LIN {X 0.311,Y -645.263,Z 996.603,A 0.000,B 0.000,C 90.000,E1 324.482} C_DIS
LIN {X 0.129,Y -646.144,Z 996.595,A 0.000,B 0.000,C 90.000,E1 323.004} C_DIS
LIN {X -0.105,Y -646.582,Z 996.589,A 0.000,B 0.000,C 90.000,E1 322.029} C_DIS
LIN {X 0.123,Y -647.178,Z 996.581,A 0.000,B 0.000,C 90.000,E1 320.517} C_DIS
LIN {X -0.362,Y -648.118,Z 996.568,A 0.000,B 0.000,C 90.000,E1 318.324} C_DIS
LIN {X 0.227,Y -649.121,Z 996.560,A 0.000,B 0.000,C 90.000,E1 316.782} C_DIS
LIN {X -0.160,Y -650.130,Z 996.550,A 0.000,B 0.000,C 90.000,E1 315.081} C_DIS
LIN {X -0.098,Y -651.626,Z 996.539,A 0.000,B 0.000,C 90.000,E1 313.095} C_DIS
LIN {X 0.087,Y -652.642,Z 996.531,A 0.000,B 0.000,C 90.000,E1 311.595} C_DIS
LIN {X -0.104,Y -653.353,Z 996.524,A 0.000,B 0.000,C 90.000,E1 310.378} C_DIS
LIN {X -0.253,Y -654.049,Z 996.516,A 0.000,B 0.000,C 90.000,E1 308.910} C_DIS
LIN {X -0.386,Y -654.669,Z 996.508,A 0.000,B 0.000,C 90.000,E1 307.443} C_DIS
LIN {X 0.072,Y -654.916,Z 996.504,A 0.000,B 0.000,C 90.000,E1 306.664} C_DIS
LIN {X 0.085,Y -655.183,Z 996.496,A 0.000,B 0.000,C 90.000,E1 305.185} C_DIS
LIN {X 0.192,Y -655.481,Z 996.486,A 0.000,B 0.000,C 90.000,E1 303.452} C_DIS
LIN {X 0.053,Y -661.224,Z 996.451,A 0.000,B 0.000,C 90.000,E1 297.078} C_DIS
LIN {X -0.315,Y -664.130,Z 996.440,A 0.000,B 0.000,C 90.000,E1 295.155} C_DIS
LIN {X -0.012,Y -665.464,Z 996.434,A 0.000,B 0.000,C 90.000,E1 294.155} C_DIS
LIN {X -0.299,Y -666.631,Z 996.429,A 0.000,B 0.000,C 90.000,E1 293.206} C_DIS
LIN {X -0.114,Y -667.165,Z 996.425,A 0.000,B 0.000,C 90.000,E1 292.461} C_DIS
LIN {X -0.071,Y -667.271,Z 996.422,A 0.000,B 0.000,C 90.000,E1 291.972} C_DIS
LIN {X 0.220,Y -666.897,Z 996.419,A 0.000,B 0.000,C 90.000,E1 291.461} C_DIS
LIN {X 0.120,Y -666.527,Z 996.418,A 0.000,B 0.000,C 90.000,E1 291.227} C_DIS
LIN {X 0.260,Y -665.623,Z 996.417,A 0.000,B 0.000,C 90.000,E1 290.972} C_DIS
LIN {X 0.229,Y -664.050,Z 996.415,A 0.000,B 0.000,C 90.000,E1 290.610} C_DIS
LIN {X 0.296,Y -663.310,Z 996.414,A 0.000,B 0.000,C 90.000,E1 290.482} C_DIS
LIN {X 0.127,Y -662.192,Z 996.413,A 0.000,B 0.000,C 90.000,E1 290.375} C_DIS
LIN {X 0.079,Y -657.367,Z 996.411,A 0.000,B 0.000,C 90.000,E1 289.939} C_DIS
LIN {X 0.198,Y -655.675,Z 996.410,A 0.000,B 0.000,C 90.000,E1 289.812} C_DIS
LIN {X 0.177,Y -647.687,Z 996.408,A 0.000,B 0.000,C 90.000,E1 289.341} C_DIS
LIN {X -0.198,Y -644.564,Z 996.407,A 0.000,B 0.000,C 90.000,E1 289.195} C_DIS
LIN {X -0.301,Y -640.203,Z 996.405,A 0.000,B 0.000,C 90.000,E1 288.906} C_DIS
LIN {X -0.336,Y -640.181,Z 996.405,A 0.000,B 0.000,C 90.000,E1 288.906} C_DIS
LIN {X -0.088,Y -640.114,Z 996.405,A 0.000,B 0.000,C 90.000,E1 288.833} C_DIS
LIN {X 0.205,Y -641.641,Z 996.402,A 0.000,B 0.000,C 90.000,E1 288.417} C_DIS
LIN {X -0.250,Y -649.985,Z 996.395,A 0.000,B 0.000,C 90.000,E1 287.094} C_DIS
LIN {X 0.135,Y -653.488,Z 996.391,A 0.000,B 0.000,C 90.000,E1 286.441} C_DIS
LIN {X -0.107,Y -655.841,Z 996.389,A 0.000,B 0.000,C 90.000,E1 285.969} C_DIS
LIN {X -0.046,Y -656.935,Z 996.387,A 0.000,B 0.000,C 90.000,E1 285.717} C_DIS
LIN {X -0.271,Y -658.778,Z 996.385,A 0.000,B 0.000,C 90.000,E1 285.245} C_DIS
LIN {X 0.258,Y -659.581,Z 996.383,A 0.000,B 0.000,C 90.000,E1 284.954} C_DIS
LIN {X 0.054,Y -660.892,Z 996.381,A 0.000,B 0.000,C 90.000,E1 284.481} C_DIS
LIN {X -0.234,Y -662.248,Z 996.376,A 0.000,B 0.000,C 90.000,E1 283.772} C_DIS
LIN {X 0.226,Y -662.891,Z 996.374,A 0.000,B 0.000,C 90.000,E1 283.244} C_DIS
LIN {X -0.045,Y -663.382,Z 996.370,A 0.000,B 0.000,C 90.000,E1 282.535} C_DIS
LIN {X 0.333,Y -663.486,Z 996.366,A 0.000,B 0.000,C 90.000,E1 281.771} C_DIS
LIN {X 0.149,Y -663.317,Z 996.363,A 0.000,B 0.000,C 90.000,E1 281.299} C_DIS
LIN {X -0.258,Y -662.702,Z 996.359,A 0.000,B 0.000,C 90.000,E1 280.602} C_DIS
LIN {X 0.200,Y -661.947,Z 996.356,A 0.000,B 0.000,C 90.000,E1 280.074} C_DIS
LIN {X -0.114,Y -660.970,Z 996.353,A 0.000,B 0.000,C 90.000,E1 279.613} C_DIS
LIN {X -0.218,Y -660.446,Z 996.352,A 0.000,B 0.000,C 90.000,E1 279.378} C_DIS
LIN {X 0.113,Y -658.986,Z 996.349,A 0.000,B 0.000,C 90.000,E1 278.859} C_DIS
LIN {X -0.211,Y -657.223,Z 996.347,A 0.000,B 0.000,C 90.000,E1 278.398} C_DIS
LIN {X 0.197,Y -655.123,Z 996.344,A 0.000,B 0.000,C 90.000,E1 277.871} C_DIS
LIN {X -0.127,Y -653.259,Z 996.342,A 0.000,B 0.000,C 90.000,E1 277.530} C_DIS
LIN {X 0.274,Y -651.156,Z 996.340,A 0.000,B 0.000,C 90.000,E1 277.125} C_DIS
LIN {X -0.098,Y -647.850,Z 996.337,A 0.000,B 0.000,C 90.000,E1 276.663} C_DIS
LIN {X 0.051,Y -643.017,Z 996.334,A 0.000,B 0.000,C 90.000,E1 276.030} C_DIS
LIN {X 0.267,Y -638.641,Z 996.331,A 0.000,B 0.000,C 90.000,E1 275.511} C_DIS
LIN {X -0.240,Y -632.519,Z 996.327,A 0.000,B 0.000,C 90.000,E1 274.935} C_DIS
LIN {X 0.180,Y -627.269,Z 996.325,A 0.000,B 0.000,C 90.000,E1 274.416} C_DIS
LIN {X 0.190,Y -618.735,Z 996.321,A 0.000,B 0.000,C 90.000,E1 273.726} C_DIS
LIN {X 0.131,Y -611.173,Z 996.318,A 0.000,B 0.000,C 90.000,E1 273.212} C_DIS
LIN {X -0.225,Y -604.977,Z 996.316,A 0.000,B 0.000,C 90.000,E1 272.865} C_DIS
LIN {X 0.210,Y -598.422,Z 996.314,A 0.000,B 0.000,C 90.000,E1 272.465} C_DIS
LIN {X -0.129,Y -591.494,Z 996.312,A 0.000,B 0.000,C 90.000,E1 272.178} C_DIS
LIN {X 0.053,Y -584.129,Z 996.311,A 0.000,B 0.000,C 90.000,E1 271.892} C_DIS
LIN {X 0.222,Y -576.582,Z 996.309,A 0.000,B 0.000,C 90.000,E1 271.661} C_DIS
LIN {X -0.030,Y -570.873,Z 996.309,A 0.000,B 0.000,C 90.000,E1 271.547} C_DIS
LIN {X -0.069,Y -564.513,Z 996.308,A 0.000,B 0.000,C 90.000,E1 271.432} C_DIS
LIN {X 0.029,Y -558.252,Z 996.308,A 0.000,B 0.000,C 90.000,E1 271.375} C_DIS
LIN {X -0.014,Y -543.150,Z 996.308,A 0.000,B 0.000,C 90.000,E1 271.375} C_DIS
LIN {X 0.138,Y -542.514,Z 996.305,A 0.000,B 0.000,C 90.000,E1 270.917} C_DIS
LIN {X 0.065,Y -540.998,Z 996.293,A 0.000,B 0.000,C 90.000,E1 268.797} C_DIS
LIN {X 0.187,Y -540.032,Z 996.286,A 0.000,B 0.000,C 90.000,E1 267.364} C_DIS
LIN {X -0.262,Y -539.190,Z 996.279,A 0.000,B 0.000,C 90.000,E1 266.274} C_DIS
LIN {X -0.088,Y -537.915,Z 996.270,A 0.000,B 0.000,C 90.000,E1 264.546} C_DIS
LIN {X 0.007,Y -536.641,Z 996.262,A 0.000,B 0.000,C 90.000,E1 263.109} C_DIS
LIN {X 0.179,Y -534.965,Z 996.252,A 0.000,B 0.000,C 90.000,E1 261.376} C_DIS
LIN {X -0.133,Y -533.227,Z 996.243,A 0.000,B 0.000,C 90.000,E1 259.690} C_DIS
LIN {X 0.183,Y -531.087,Z 996.232,A 0.000,B 0.000,C 90.000,E1 257.645} C_DIS
LIN {X 0.036,Y -528.840,Z 996.220,A 0.000,B 0.000,C 90.000,E1 255.644} C_DIS
LIN {X 0.126,Y -525.952,Z 996.206,A 0.000,B 0.000,C 90.000,E1 253.032} C_DIS
LIN {X 0.117,Y -524.641,Z 996.199,A 0.000,B 0.000,C 90.000,E1 251.873} C_DIS
LIN {X -0.069,Y -523.224,Z 996.193,A 0.000,B 0.000,C 90.000,E1 250.732} C_DIS
LIN {X 0.205,Y -521.009,Z 996.183,A 0.000,B 0.000,C 90.000,E1 248.954} C_DIS
LIN {X -0.054,Y -518.737,Z 996.174,A 0.000,B 0.000,C 90.000,E1 247.230} C_DIS
LIN {X -0.105,Y -517.539,Z 996.169,A 0.000,B 0.000,C 90.000,E1 246.357} C_DIS
LIN {X 0.305,Y -515.339,Z 996.160,A 0.000,B 0.000,C 90.000,E1 244.845} C_DIS
LIN {X 0.092,Y -513.544,Z 996.154,A 0.000,B 0.000,C 90.000,E1 243.691} C_DIS
LIN {X -0.059,Y -510.285,Z 996.142,A 0.000,B 0.000,C 90.000,E1 241.641} C_DIS
LIN {X 0.221,Y -507.774,Z 996.134,A 0.000,B 0.000,C 90.000,E1 240.127} C_DIS
LIN {X 0.129,Y -505.635,Z 996.128,A 0.000,B 0.000,C 90.000,E1 238.948} C_DIS
LIN {X 0.142,Y -502.701,Z 996.119,A 0.000,B 0.000,C 90.000,E1 237.454} C_DIS
LIN {X -0.193,Y -500.193,Z 996.113,A 0.000,B 0.000,C 90.000,E1 236.294} C_DIS
LIN {X 0.126,Y -497.517,Z 996.106,A 0.000,B 0.000,C 90.000,E1 235.055} C_DIS
LIN {X -0.272,Y -495.439,Z 996.101,A 0.000,B 0.000,C 90.000,E1 234.196} C_DIS
LIN {X 0.108,Y -491.665,Z 996.093,A 0.000,B 0.000,C 90.000,E1 232.637} C_DIS
LIN {X -0.008,Y -486.585,Z 996.081,A 0.000,B 0.000,C 90.000,E1 230.517} C_DIS
LIN {X 0.001,Y -481.585,Z 996.069,A 0.000,B 0.000,C 90.000,E1 228.366} C_DIS
LIN {X 0.107,Y -475.618,Z 996.053,A 0.000,B 0.000,C 90.000,E1 225.567} C_DIS
LIN {X -0.146,Y -473.022,Z 996.046,A 0.000,B 0.000,C 90.000,E1 224.352} C_DIS
LIN {X -0.011,Y -469.581,Z 996.038,A 0.000,B 0.000,C 90.000,E1 222.771} C_DIS
LIN {X 0.155,Y -465.426,Z 996.027,A 0.000,B 0.000,C 90.000,E1 220.862} C_DIS
LIN {X 0.024,Y -463.299,Z 996.022,A 0.000,B 0.000,C 90.000,E1 219.930} C_DIS
LIN {X 0.066,Y -459.757,Z 996.013,A 0.000,B 0.000,C 90.000,E1 218.338} C_DIS
LIN {X 0.052,Y -455.563,Z 996.002,A 0.000,B 0.000,C 90.000,E1 216.423} C_DIS
LIN {X 0.130,Y -451.324,Z 995.992,A 0.000,B 0.000,C 90.000,E1 214.485} C_DIS
LIN {X 0.040,Y -447.850,Z 995.983,A 0.000,B 0.000,C 90.000,E1 212.880} C_DIS
LIN {X 0.072,Y -443.624,Z 995.972,A 0.000,B 0.000,C 90.000,E1 210.924} C_DIS
LIN {X 0.116,Y -440.040,Z 995.963,A 0.000,B 0.000,C 90.000,E1 209.283} C_DIS
LIN {X -0.048,Y -434.074,Z 995.948,A 0.000,B 0.000,C 90.000,E1 206.668} C_DIS
LIN {X -0.198,Y -430.307,Z 995.939,A 0.000,B 0.000,C 90.000,E1 205.027} C_DIS
LIN {X 0.131,Y -425.028,Z 995.926,A 0.000,B 0.000,C 90.000,E1 202.642} C_DIS
LIN {X 0.026,Y -421.297,Z 995.917,A 0.000,B 0.000,C 90.000,E1 200.972} C_DIS
LIN {X 0.092,Y -417.787,Z 995.907,A 0.000,B 0.000,C 90.000,E1 199.268} C_DIS
LIN {X -0.144,Y -413.191,Z 995.894,A 0.000,B 0.000,C 90.000,E1 196.913} C_DIS
LIN {X -0.092,Y -410.150,Z 995.884,A 0.000,B 0.000,C 90.000,E1 195.190} C_DIS
LIN {X -0.092,Y -406.672,Z 995.873,A 0.000,B 0.000,C 90.000,E1 193.119} C_DIS
LIN {X 0.120,Y -403.177,Z 995.861,A 0.000,B 0.000,C 90.000,E1 191.007} C_DIS
LIN {X 0.063,Y -398.744,Z 995.846,A 0.000,B 0.000,C 90.000,E1 188.219} C_DIS
LIN {X -0.028,Y -397.918,Z 995.842,A 0.000,B 0.000,C 90.000,E1 187.530} C_DIS
LIN {X -0.039,Y -397.792,Z 995.840,A 0.000,B 0.000,C 90.000,E1 187.182} C_DIS
LIN {X -0.063,Y -397.525,Z 995.838,A 0.000,B 0.000,C 90.000,E1 186.834} C_DIS
LIN {X -0.187,Y -397.605,Z 995.832,A 0.000,B 0.000,C 90.000,E1 185.796} C_DIS
LIN {X -0.159,Y -398.314,Z 995.829,A 0.000,B 0.000,C 90.000,E1 185.220} C_DIS
LIN {X -0.135,Y -400.044,Z 995.825,A 0.000,B 0.000,C 90.000,E1 184.531} C_DIS
LIN {X 0.212,Y -401.987,Z 995.822,A 0.000,B 0.000,C 90.000,E1 183.955} C_DIS
LIN {X 0.194,Y -405.588,Z 995.819,A 0.000,B 0.000,C 90.000,E1 183.326} C_DIS
LIN {X 0.175,Y -406.659,Z 995.818,A 0.000,B 0.000,C 90.000,E1 183.154} C_DIS
LIN {X -0.137,Y -412.804,Z 995.813,A 0.000,B 0.000,C 90.000,E1 182.407} C_DIS
LIN {X 0.158,Y -420.075,Z 995.809,A 0.000,B 0.000,C 90.000,E1 181.547} C_DIS
LIN {X 0.147,Y -435.791,Z 995.799,A 0.000,B 0.000,C 90.000,E1 179.885} C_DIS
LIN {X -0.131,Y -444.377,Z 995.795,A 0.000,B 0.000,C 90.000,E1 179.026} C_DIS
LIN {X -0.213,Y -452.675,Z 995.790,A 0.000,B 0.000,C 90.000,E1 178.165} C_DIS
LIN {X 0.040,Y -460.720,Z 995.785,A 0.000,B 0.000,C 90.000,E1 177.249} C_DIS
LIN {X 0.043,Y -468.718,Z 995.780,A 0.000,B 0.000,C 90.000,E1 176.331} C_DIS
LIN {X -0.013,Y -473.533,Z 995.776,A 0.000,B 0.000,C 90.000,E1 175.755} C_DIS
LIN {X -0.019,Y -482.215,Z 995.770,A 0.000,B 0.000,C 90.000,E1 174.666} C_DIS
LIN {X -0.021,Y -488.963,Z 995.765,A 0.000,B 0.000,C 90.000,E1 173.742} C_DIS
LIN {X 0.223,Y -496.573,Z 995.759,A 0.000,B 0.000,C 90.000,E1 172.648} C_DIS
LIN {X -0.001,Y -506.023,Z 995.752,A 0.000,B 0.000,C 90.000,E1 171.319} C_DIS
LIN {X -0.190,Y -513.971,Z 995.745,A 0.000,B 0.000,C 90.000,E1 170.151} C_DIS
LIN {X -0.047,Y -523.949,Z 995.736,A 0.000,B 0.000,C 90.000,E1 168.522} C_DIS
LIN {X -0.186,Y -530.219,Z 995.731,A 0.000,B 0.000,C 90.000,E1 167.521} C_DIS
LIN {X -0.190,Y -537.923,Z 995.723,A 0.000,B 0.000,C 90.000,E1 166.228} C_DIS
LIN {X -0.226,Y -546.298,Z 995.716,A 0.000,B 0.000,C 90.000,E1 164.810} C_DIS
LIN {X 0.059,Y -551.904,Z 995.710,A 0.000,B 0.000,C 90.000,E1 163.795} C_DIS
LIN {X 0.016,Y -556.691,Z 995.705,A 0.000,B 0.000,C 90.000,E1 162.960} C_DIS
LIN {X 0.212,Y -563.363,Z 995.698,A 0.000,B 0.000,C 90.000,E1 161.692} C_DIS
LIN {X -0.153,Y -566.952,Z 995.695,A 0.000,B 0.000,C 90.000,E1 161.040} C_DIS
LIN {X 0.042,Y -572.002,Z 995.689,A 0.000,B 0.000,C 90.000,E1 160.061} C_DIS
LIN {X -0.066,Y -578.070,Z 995.682,A 0.000,B 0.000,C 90.000,E1 158.847} C_DIS
LIN {X 0.162,Y -580.612,Z 995.680,A 0.000,B 0.000,C 90.000,E1 158.284} C_DIS
LIN {X -0.080,Y -585.418,Z 995.674,A 0.000,B 0.000,C 90.000,E1 157.230} C_DIS
LIN {X 0.088,Y -588.949,Z 995.669,A 0.000,B 0.000,C 90.000,E1 156.410} C_DIS
LIN {X 0.053,Y -592.211,Z 995.665,A 0.000,B 0.000,C 90.000,E1 155.613} C_DIS
LIN {X -0.247,Y -595.193,Z 995.660,A 0.000,B 0.000,C 90.000,E1 154.845} C_DIS
LIN {X 0.024,Y -597.992,Z 995.656,A 0.000,B 0.000,C 90.000,E1 154.024} C_DIS
LIN {X -0.215,Y -600.502,Z 995.651,A 0.000,B 0.000,C 90.000,E1 153.256} C_DIS
LIN {X 0.319,Y -603.785,Z 995.646,A 0.000,B 0.000,C 90.000,E1 152.153} C_DIS
LIN {X 0.078,Y -606.853,Z 995.640,A 0.000,B 0.000,C 90.000,E1 151.129} C_DIS
LIN {X -0.147,Y -611.419,Z 995.631,A 0.000,B 0.000,C 90.000,E1 149.587} C_DIS
LIN {X -0.035,Y -615.071,Z 995.624,A 0.000,B 0.000,C 90.000,E1 148.280} C_DIS
LIN {X 0.234,Y -619.297,Z 995.615,A 0.000,B 0.000,C 90.000,E1 146.707} C_DIS
LIN {X -0.125,Y -625.066,Z 995.604,A 0.000,B 0.000,C 90.000,E1 144.689} C_DIS
LIN {X 0.198,Y -629.354,Z 995.595,A 0.000,B 0.000,C 90.000,E1 143.130} C_DIS
LIN {X 0.101,Y -633.551,Z 995.587,A 0.000,B 0.000,C 90.000,E1 141.618} C_DIS
LIN {X 0.099,Y -637.020,Z 995.580,A 0.000,B 0.000,C 90.000,E1 140.356} C_DIS
LIN {X 0.152,Y -640.427,Z 995.573,A 0.000,B 0.000,C 90.000,E1 139.094} C_DIS
LIN {X 0.202,Y -643.771,Z 995.566,A 0.000,B 0.000,C 90.000,E1 137.838} C_DIS
LIN {X -0.373,Y -650.026,Z 995.553,A 0.000,B 0.000,C 90.000,E1 135.648} C_DIS
LIN {X 0.176,Y -656.166,Z 995.542,A 0.000,B 0.000,C 90.000,E1 133.623} C_DIS
LIN {X 0.004,Y -661.911,Z 995.533,A 0.000,B 0.000,C 90.000,E1 131.919} C_DIS
LIN {X -0.020,Y -666.158,Z 995.526,A 0.000,B 0.000,C 90.000,E1 130.701} C_DIS
LIN {X -0.410,Y -671.080,Z 995.518,A 0.000,B 0.000,C 90.000,E1 129.277} C_DIS
LIN {X 0.221,Y -674.784,Z 995.511,A 0.000,B 0.000,C 90.000,E1 128.016} C_DIS
LIN {X 0.098,Y -679.086,Z 995.503,A 0.000,B 0.000,C 90.000,E1 126.583} C_DIS
LIN {X 0.051,Y -683.153,Z 995.495,A 0.000,B 0.000,C 90.000,E1 125.152} C_DIS
LIN {X -0.331,Y -686.478,Z 995.489,A 0.000,B 0.000,C 90.000,E1 123.992} C_DIS
LIN {X 0.151,Y -690.700,Z 995.479,A 0.000,B 0.000,C 90.000,E1 122.291} C_DIS
LIN {X -0.107,Y -693.781,Z 995.473,A 0.000,B 0.000,C 90.000,E1 121.131} C_DIS
LIN {X 0.022,Y -695.510,Z 995.469,A 0.000,B 0.000,C 90.000,E1 120.413} C_DIS
LIN {X 0.168,Y -697.410,Z 995.464,A 0.000,B 0.000,C 90.000,E1 119.461} C_DIS
LIN {X 0.333,Y -698.629,Z 995.460,A 0.000,B 0.000,C 90.000,E1 118.743} C_DIS
LIN {X -0.435,Y -699.539,Z 995.456,A 0.000,B 0.000,C 90.000,E1 118.103} C_DIS
LIN {X -0.247,Y -700.219,Z 995.452,A 0.000,B 0.000,C 90.000,E1 117.385} C_DIS
LIN {X -0.175,Y -701.441,Z 995.444,A 0.000,B 0.000,C 90.000,E1 115.976} C_DIS
LIN {X -0.282,Y -701.956,Z 995.440,A 0.000,B 0.000,C 90.000,E1 115.283} C_DIS
LIN {X -0.104,Y -702.267,Z 995.435,A 0.000,B 0.000,C 90.000,E1 114.335} C_DIS
LIN {X 0.173,Y -702.193,Z 995.434,A 0.000,B 0.000,C 90.000,E1 114.079} C_DIS
LIN {X -0.202,Y -701.685,Z 995.431,A 0.000,B 0.000,C 90.000,E1 113.643} C_DIS
LIN {X 0.072,Y -700.992,Z 995.430,A 0.000,B 0.000,C 90.000,E1 113.387} C_DIS
LIN {X -0.308,Y -698.825,Z 995.427,A 0.000,B 0.000,C 90.000,E1 112.950} C_DIS
LIN {X -0.175,Y -698.084,Z 995.427,A 0.000,B 0.000,C 90.000,E1 112.823} C_DIS
LIN {X -0.044,Y -696.980,Z 995.426,A 0.000,B 0.000,C 90.000,E1 112.695} C_DIS
LIN {X 0.417,Y -691.563,Z 995.424,A 0.000,B 0.000,C 90.000,E1 112.206} C_DIS
LIN {X -0.213,Y -689.627,Z 995.423,A 0.000,B 0.000,C 90.000,E1 112.153} C_DIS
LIN {X -0.037,Y -684.985,Z 995.422,A 0.000,B 0.000,C 90.000,E1 111.972} C_DIS
LIN {X 0.127,Y -682.156,Z 995.422,A 0.000,B 0.000,C 90.000,E1 111.897} C_DIS
LIN {X 0.152,Y -675.748,Z 995.421,A 0.000,B 0.000,C 90.000,E1 111.791} C_DIS
LIN {X 0.299,Y -674.808,Z 995.421,A 0.000,B 0.000,C 90.000,E1 111.770} C_DIS
LIN {X 0.227,Y -619.713,Z 995.421,A 0.000,B 0.000,C 90.000,E1 111.770} C_DIS
LIN {X 0.231,Y -616.938,Z 995.421,A 0.000,B 0.000,C 90.000,E1 111.716} C_DIS
LIN {X 0.233,Y -610.485,Z 995.420,A 0.000,B 0.000,C 90.000,E1 111.535} C_DIS
LIN {X 0.093,Y -602.550,Z 995.418,A 0.000,B 0.000,C 90.000,E1 111.227} C_DIS
LIN {X 0.175,Y -599.234,Z 995.417,A 0.000,B 0.000,C 90.000,E1 111.046} C_DIS
LIN {X 0.039,Y -594.664,Z 995.416,A 0.000,B 0.000,C 90.000,E1 110.791} C_DIS
LIN {X 0.206,Y -589.016,Z 995.413,A 0.000,B 0.000,C 90.000,E1 110.375} C_DIS
LIN {X -0.067,Y -577.729,Z 995.408,A 0.000,B 0.000,C 90.000,E1 109.504} C_DIS
LIN {X 0.142,Y -573.374,Z 995.406,A 0.000,B 0.000,C 90.000,E1 109.141} C_DIS
LIN {X 0.154,Y -566.545,Z 995.404,A 0.000,B 0.000,C 90.000,E1 108.725} C_DIS
LIN {X -0.062,Y -564.936,Z 995.404,A 0.000,B 0.000,C 90.000,E1 108.652} C_DIS
LIN {X 0.003,Y -550.927,Z 995.400,A 0.000,B 0.000,C 90.000,E1 107.946} C_DIS
LIN {X -0.085,Y -549.106,Z 995.399,A 0.000,B 0.000,C 90.000,E1 107.764} C_DIS
LIN {X -0.126,Y -549.097,Z 995.399,A 0.000,B 0.000,C 90.000,E1 107.764} C_DIS
LIN {X -0.094,Y -548.641,Z 995.397,A 0.000,B 0.000,C 90.000,E1 107.457} C_DIS
LIN {X 0.113,Y -548.754,Z 995.393,A 0.000,B 0.000,C 90.000,E1 106.732} C_DIS
LIN {X 0.122,Y -549.258,Z 995.387,A 0.000,B 0.000,C 90.000,E1 105.607} C_DIS
LIN {X 0.174,Y -550.410,Z 995.374,A 0.000,B 0.000,C 90.000,E1 103.355} C_DIS
LIN {X 0.092,Y -553.910,Z 995.353,A 0.000,B 0.000,C 90.000,E1 99.443} C_DIS
LIN {X 0.083,Y -555.388,Z 995.345,A 0.000,B 0.000,C 90.000,E1 98.049} C_DIS
LIN {X -0.040,Y -556.595,Z 995.339,A 0.000,B 0.000,C 90.000,E1 96.947} C_DIS
LIN {X -0.218,Y -557.646,Z 995.332,A 0.000,B 0.000,C 90.000,E1 95.853} C_DIS
LIN {X 0.250,Y -558.637,Z 995.325,A 0.000,B 0.000,C 90.000,E1 94.416} C_DIS
LIN {X 0.178,Y -559.498,Z 995.317,A 0.000,B 0.000,C 90.000,E1 93.037} C_DIS
LIN {X 0.083,Y -560.229,Z 995.309,A 0.000,B 0.000,C 90.000,E1 91.661} C_DIS
LIN {X 0.183,Y -561.183,Z 995.299,A 0.000,B 0.000,C 90.000,E1 89.714} C_DIS
LIN {X 0.010,Y -561.645,Z 995.292,A 0.000,B 0.000,C 90.000,E1 88.625} C_DIS
LIN {X -0.046,Y -561.934,Z 995.285,A 0.000,B 0.000,C 90.000,E1 87.249} C_DIS
LIN {X 0.033,Y -562.193,Z 995.276,A 0.000,B 0.000,C 90.000,E1 85.584} C_DIS
LIN {X -0.157,Y -562.522,Z 995.263,A 0.000,B 0.000,C 90.000,E1 83.394} C_DIS
LIN {X 0.132,Y -562.915,Z 995.253,A 0.000,B 0.000,C 90.000,E1 81.432} C_DIS
LIN {X 0.206,Y -563.660,Z 995.240,A 0.000,B 0.000,C 90.000,E1 79.218} C_DIS
LIN {X -0.196,Y -564.277,Z 995.233,A 0.000,B 0.000,C 90.000,E1 77.881} C_DIS
LIN {X 0.036,Y -564.902,Z 995.227,A 0.000,B 0.000,C 90.000,E1 76.756} C_DIS
LIN {X 0.019,Y -566.527,Z 995.213,A 0.000,B 0.000,C 90.000,E1 74.283} C_DIS
LIN {X 0.011,Y -567.918,Z 995.202,A 0.000,B 0.000,C 90.000,E1 72.362} C_DIS
LIN {X 0.261,Y -568.884,Z 995.194,A 0.000,B 0.000,C 90.000,E1 70.967} C_DIS
LIN {X 0.183,Y -569.600,Z 995.188,A 0.000,B 0.000,C 90.000,E1 69.880} C_DIS
LIN {X -0.080,Y -570.393,Z 995.181,A 0.000,B 0.000,C 90.000,E1 68.539} C_DIS
LIN {X -0.297,Y -571.201,Z 995.172,A 0.000,B 0.000,C 90.000,E1 66.922} C_DIS
LIN {X -0.095,Y -571.774,Z 995.164,A 0.000,B 0.000,C 90.000,E1 65.537} C_DIS
LIN {X 0.280,Y -572.182,Z 995.158,A 0.000,B 0.000,C 90.000,E1 64.409} C_DIS
LIN {X -0.027,Y -572.648,Z 995.150,A 0.000,B 0.000,C 90.000,E1 63.076} C_DIS
LIN {X 0.040,Y -573.059,Z 995.141,A 0.000,B 0.000,C 90.000,E1 61.435} C_DIS
LIN {X 0.004,Y -573.412,Z 995.134,A 0.000,B 0.000,C 90.000,E1 60.078} C_DIS
LIN {X -0.113,Y -573.660,Z 995.125,A 0.000,B 0.000,C 90.000,E1 58.456} C_DIS
LIN {X -0.218,Y -573.869,Z 995.116,A 0.000,B 0.000,C 90.000,E1 56.834} C_DIS
LIN {X -0.153,Y -574.007,Z 995.108,A 0.000,B 0.000,C 90.000,E1 55.468} C_DIS
LIN {X 0.279,Y -573.985,Z 995.104,A 0.000,B 0.000,C 90.000,E1 54.609} C_DIS
LIN {X 0.060,Y -573.837,Z 995.098,A 0.000,B 0.000,C 90.000,E1 53.543} C_DIS
LIN {X -0.162,Y -573.463,Z 995.091,A 0.000,B 0.000,C 90.000,E1 52.477} C_DIS
LIN {X 0.100,Y -572.771,Z 995.084,A 0.000,B 0.000,C 90.000,E1 51.090} C_DIS
LIN {X 0.208,Y -572.037,Z 995.078,A 0.000,B 0.000,C 90.000,E1 49.989} C_DIS
LIN {X -0.009,Y -570.820,Z 995.070,A 0.000,B 0.000,C 90.000,E1 48.647} C_DIS
LIN {X -0.111,Y -569.940,Z 995.066,A 0.000,B 0.000,C 90.000,E1 47.838} C_DIS
LIN {X 0.204,Y -568.885,Z 995.061,A 0.000,B 0.000,C 90.000,E1 46.986} C_DIS
LIN {X 0.197,Y -567.136,Z 995.055,A 0.000,B 0.000,C 90.000,E1 45.891} C_DIS
LIN {X 0.070,Y -565.627,Z 995.051,A 0.000,B 0.000,C 90.000,E1 45.081} C_DIS
LIN {X -0.389,Y -563.322,Z 995.044,A 0.000,B 0.000,C 90.000,E1 44.028} C_DIS
LIN {X -0.149,Y -561.311,Z 995.040,A 0.000,B 0.000,C 90.000,E1 43.176} C_DIS
LIN {X 0.072,Y -558.994,Z 995.035,A 0.000,B 0.000,C 90.000,E1 42.324} C_DIS
LIN {X -0.149,Y -556.420,Z 995.031,A 0.000,B 0.000,C 90.000,E1 41.515} C_DIS
LIN {X 0.010,Y -553.586,Z 995.026,A 0.000,B 0.000,C 90.000,E1 40.663} C_DIS
LIN {X 0.202,Y -550.359,Z 995.021,A 0.000,B 0.000,C 90.000,E1 39.806} C_DIS
LIN {X 0.090,Y -547.356,Z 995.017,A 0.000,B 0.000,C 90.000,E1 39.116} C_DIS
LIN {X 0.030,Y -544.139,Z 995.013,A 0.000,B 0.000,C 90.000,E1 38.418} C_DIS
LIN {X -0.121,Y -539.391,Z 995.008,A 0.000,B 0.000,C 90.000,E1 37.443} C_DIS
LIN {X -0.073,Y -533.459,Z 995.002,A 0.000,B 0.000,C 90.000,E1 36.297} C_DIS
LIN {X -0.096,Y -528.719,Z 994.997,A 0.000,B 0.000,C 90.000,E1 35.438} C_DIS
LIN {X 0.288,Y -525.351,Z 994.994,A 0.000,B 0.000,C 90.000,E1 34.818} C_DIS
LIN {X -0.004,Y -519.078,Z 994.988,A 0.000,B 0.000,C 90.000,E1 33.833} C_DIS
LIN {X 0.021,Y -515.306,Z 994.985,A 0.000,B 0.000,C 90.000,E1 33.245} C_DIS
LIN {X -0.128,Y -511.247,Z 994.982,A 0.000,B 0.000,C 90.000,E1 32.673} C_DIS
LIN {X -0.037,Y -507.057,Z 994.978,A 0.000,B 0.000,C 90.000,E1 32.084} C_DIS
LIN {X 0.177,Y -502.435,Z 994.975,A 0.000,B 0.000,C 90.000,E1 31.465} C_DIS
LIN {X 0.092,Y -497.534,Z 994.972,A 0.000,B 0.000,C 90.000,E1 30.875} C_DIS
LIN {X -0.238,Y -493.592,Z 994.969,A 0.000,B 0.000,C 90.000,E1 30.463} C_DIS
LIN {X 0.278,Y -486.763,Z 994.965,A 0.000,B 0.000,C 90.000,E1 29.667} C_DIS
LIN {X -0.112,Y -476.948,Z 994.960,A 0.000,B 0.000,C 90.000,E1 28.743} C_DIS
LIN {X -0.030,Y -471.198,Z 994.957,A 0.000,B 0.000,C 90.000,E1 28.180} C_DIS
LIN {X -0.187,Y -462.401,Z 994.952,A 0.000,B 0.000,C 90.000,E1 27.385} C_DIS
LIN {X 0.010,Y -451.858,Z 994.947,A 0.000,B 0.000,C 90.000,E1 26.437} C_DIS
LIN {X -0.116,Y -439.624,Z 994.941,A 0.000,B 0.000,C 90.000,E1 25.412} C_DIS
LIN {X 0.189,Y -421.796,Z 994.932,A 0.000,B 0.000,C 90.000,E1 23.770} C_DIS
LIN {X 0.205,Y -407.446,Z 994.924,A 0.000,B 0.000,C 90.000,E1 22.333} C_DIS
LIN {X -0.147,Y -399.082,Z 994.919,A 0.000,B 0.000,C 90.000,E1 21.461} C_DIS
LIN {X 0.209,Y -395.627,Z 994.917,A 0.000,B 0.000,C 90.000,E1 20.972} C_DIS
LIN {X -0.079,Y -392.370,Z 994.913,A 0.000,B 0.000,C 90.000,E1 20.429} C_DIS
LIN {X 0.001,Y -390.730,Z 994.911,A 0.000,B 0.000,C 90.000,E1 19.885} C_DIS
LIN {X -0.039,Y -390.135,Z 994.907,A 0.000,B 0.000,C 90.000,E1 19.268} C_DIS
LIN {X 0.025,Y -390.287,Z 994.904,A 0.000,B 0.000,C 90.000,E1 18.725} C_DIS
LIN {X -0.062,Y -394.095,Z 994.882,A 0.000,B 0.000,C 90.000,E1 14.828} C_DIS
LIN {X -0.088,Y -399.215,Z 994.861,A 0.000,B 0.000,C 90.000,E1 10.950} C_DIS
LIN {X 0.221,Y -405.140,Z 994.841,A 0.000,B 0.000,C 90.000,E1 7.409} C_DIS
LIN {X 0.174,Y -412.109,Z 994.822,A 0.000,B 0.000,C 90.000,E1 3.955} C_DIS
LIN {X 0.194,Y -415.137,Z 994.815,A 0.000,B 0.000,C 90.000,E1 2.579} C_DIS
LIN {X -0.171,Y -417.369,Z 994.809,A 0.000,B 0.000,C 90.000,E1 1.604} C_DIS
LIN {X -0.129,Y -419.629,Z 994.805,A 0.000,B 0.000,C 90.000,E1 0.917} C_DIS
LIN {X -0.067,Y -423.062,Z 994.801,A 0.000,B 0.000,C 90.000,E1 0.229} C_DIS
LIN {X 0.000,Y -425.018,Z 994.800,A 0.000,B 0.000,C 90.000,E1 360.000} C_DIS
LIN {X -0.089,Y -428.580,Z 994.798,A 0.000,B 0.000,C 90.000,E1 359.656} C_DIS
LIN {X 0.129,Y -434.164,Z 994.796,A 0.000,B 0.000,C 90.000,E1 359.255} C_DIS
LIN {X -0.091,Y -452.151,Z 994.790,A 0.000,B 0.000,C 90.000,E1 358.282} C_DIS
LIN {X -0.077,Y -467.193,Z 994.786,A 0.000,B 0.000,C 90.000,E1 357.421} C_DIS
LIN {X -0.022,Y -485.328,Z 994.780,A 0.000,B 0.000,C 90.000,E1 356.388} C_DIS
LIN {X -0.199,Y -498.518,Z 994.776,A 0.000,B 0.000,C 90.000,E1 355.641} C_DIS
LIN {X -0.244,Y -509.669,Z 994.772,A 0.000,B 0.000,C 90.000,E1 354.951} C_DIS
LIN {X -0.218,Y -518.921,Z 994.768,A 0.000,B 0.000,C 90.000,E1 354.318} C_DIS
LIN {X -0.048,Y -526.570,Z 994.765,A 0.000,B 0.000,C 90.000,E1 353.742} C_DIS
LIN {X -0.090,Y -533.940,Z 994.762,A 0.000,B 0.000,C 90.000,E1 353.166} C_DIS
LIN {X -0.254,Y -540.716,Z 994.759,A 0.000,B 0.000,C 90.000,E1 352.591} C_DIS
LIN {X 0.188,Y -547.373,Z 994.755,A 0.000,B 0.000,C 90.000,E1 351.894} C_DIS
LIN {X -0.097,Y -553.780,Z 994.751,A 0.000,B 0.000,C 90.000,E1 351.254} C_DIS
LIN {X 0.108,Y -558.537,Z 994.748,A 0.000,B 0.000,C 90.000,E1 350.679} C_DIS
LIN {X -0.161,Y -562.958,Z 994.745,A 0.000,B 0.000,C 90.000,E1 350.151} C_DIS
LIN {X -0.085,Y -567.889,Z 994.741,A 0.000,B 0.000,C 90.000,E1 349.454} C_DIS
LIN {X 0.275,Y -571.477,Z 994.738,A 0.000,B 0.000,C 90.000,E1 348.870} C_DIS
LIN {X -0.049,Y -577.928,Z 994.732,A 0.000,B 0.000,C 90.000,E1 347.813} C_DIS
LIN {X -0.054,Y -585.002,Z 994.725,A 0.000,B 0.000,C 90.000,E1 346.464} C_DIS
LIN {X 0.112,Y -589.014,Z 994.720,A 0.000,B 0.000,C 90.000,E1 345.644} C_DIS
LIN {X 0.090,Y -594.775,Z 994.714,A 0.000,B 0.000,C 90.000,E1 344.448} C_DIS
LIN {X -0.012,Y -600.103,Z 994.707,A 0.000,B 0.000,C 90.000,E1 343.268} C_DIS
LIN {X 0.078,Y -605.507,Z 994.700,A 0.000,B 0.000,C 90.000,E1 341.945} C_DIS
LIN {X 0.218,Y -608.753,Z 994.695,A 0.000,B 0.000,C 90.000,E1 341.148} C_DIS
LIN {X -0.121,Y -613.615,Z 994.688,A 0.000,B 0.000,C 90.000,E1 339.880} C_DIS
LIN {X 0.151,Y -615.414,Z 994.685,A 0.000,B 0.000,C 90.000,E1 339.337} C_DIS
LIN {X 0.102,Y -620.345,Z 994.677,A 0.000,B 0.000,C 90.000,E1 337.794} C_DIS
LIN {X -0.179,Y -624.121,Z 994.670,A 0.000,B 0.000,C 90.000,E1 336.538} C_DIS
LIN {X 0.166,Y -626.964,Z 994.664,A 0.000,B 0.000,C 90.000,E1 335.485} C_DIS
LIN {X 0.216,Y -628.942,Z 994.660,A 0.000,B 0.000,C 90.000,E1 334.717} C_DIS
LIN {X 0.043,Y -631.422,Z 994.654,A 0.000,B 0.000,C 90.000,E1 333.717} C_DIS
LIN {X 0.138,Y -633.060,Z 994.650,A 0.000,B 0.000,C 90.000,E1 332.948} C_DIS
LIN {X 0.115,Y -636.119,Z 994.641,A 0.000,B 0.000,C 90.000,E1 331.435} C_DIS
LIN {X -0.252,Y -637.993,Z 994.636,A 0.000,B 0.000,C 90.000,E1 330.461} C_DIS
LIN {X 0.218,Y -639.365,Z 994.632,A 0.000,B 0.000,C 90.000,E1 329.665} C_DIS
LIN {X 0.263,Y -641.327,Z 994.625,A 0.000,B 0.000,C 90.000,E1 328.408} C_DIS
LIN {X 0.218,Y -642.356,Z 994.620,A 0.000,B 0.000,C 90.000,E1 327.661} C_DIS
LIN {X 0.106,Y -643.914,Z 994.614,A 0.000,B 0.000,C 90.000,E1 326.421} C_DIS
LIN {X -0.030,Y -644.919,Z 994.608,A 0.000,B 0.000,C 90.000,E1 325.435} C_DIS
LIN {X 0.379,Y -645.756,Z 994.602,A 0.000,B 0.000,C 90.000,E1 324.402} C_DIS
LIN {X -0.214,Y -646.531,Z 994.596,A 0.000,B 0.000,C 90.000,E1 323.210} C_DIS
LIN {X 0.068,Y -647.045,Z 994.590,A 0.000,B 0.000,C 90.000,E1 322.190} C_DIS
LIN {X 0.226,Y -647.728,Z 994.580,A 0.000,B 0.000,C 90.000,E1 320.436} C_DIS
LIN {X -0.176,Y -648.550,Z 994.569,A 0.000,B 0.000,C 90.000,E1 318.485} C_DIS
LIN {X 0.306,Y -649.867,Z 994.558,A 0.000,B 0.000,C 90.000,E1 316.458} C_DIS
LIN {X -0.111,Y -651.104,Z 994.547,A 0.000,B 0.000,C 90.000,E1 314.514} C_DIS
LIN {X 0.069,Y -652.265,Z 994.539,A 0.000,B 0.000,C 90.000,E1 313.014} C_DIS
LIN {X 0.314,Y -653.147,Z 994.532,A 0.000,B 0.000,C 90.000,E1 311.757} C_DIS
LIN {X 0.083,Y -654.030,Z 994.524,A 0.000,B 0.000,C 90.000,E1 310.297} C_DIS
LIN {X -0.110,Y -654.865,Z 994.514,A 0.000,B 0.000,C 90.000,E1 308.588} C_DIS
LIN {X 0.283,Y -655.463,Z 994.506,A 0.000,B 0.000,C 90.000,E1 307.076} C_DIS
LIN {X 0.294,Y -655.689,Z 994.501,A 0.000,B 0.000,C 90.000,E1 306.091} C_DIS
LIN {X -0.142,Y -655.852,Z 994.494,A 0.000,B 0.000,C 90.000,E1 304.898} C_DIS
LIN {X -0.120,Y -656.164,Z 994.486,A 0.000,B 0.000,C 90.000,E1 303.420} C_DIS
LIN {X 0.324,Y -661.956,Z 994.450,A 0.000,B 0.000,C 90.000,E1 297.001} C_DIS
LIN {X -0.179,Y -664.553,Z 994.441,A 0.000,B 0.000,C 90.000,E1 295.335} C_DIS
LIN {X 0.126,Y -665.995,Z 994.435,A 0.000,B 0.000,C 90.000,E1 294.335} C_DIS
LIN {X -0.157,Y -667.213,Z 994.430,A 0.000,B 0.000,C 90.000,E1 293.387} C_DIS
LIN {X 0.031,Y -667.927,Z 994.426,A 0.000,B 0.000,C 90.000,E1 292.642} C_DIS
LIN {X 0.077,Y -668.103,Z 994.423,A 0.000,B 0.000,C 90.000,E1 292.153} C_DIS
LIN {X 0.227,Y -668.140,Z 994.422,A 0.000,B 0.000,C 90.000,E1 291.897} C_DIS
LIN {X 0.277,Y -667.656,Z 994.419,A 0.000,B 0.000,C 90.000,E1 291.408} C_DIS
LIN {X 0.180,Y -667.246,Z 994.418,A 0.000,B 0.000,C 90.000,E1 291.173} C_DIS
LIN {X -0.324,Y -664.486,Z 994.414,A 0.000,B 0.000,C 90.000,E1 290.610} C_DIS
LIN {X -0.256,Y -663.667,Z 994.414,A 0.000,B 0.000,C 90.000,E1 290.482} C_DIS
LIN {X -0.192,Y -662.435,Z 994.413,A 0.000,B 0.000,C 90.000,E1 290.355} C_DIS
LIN {X -0.080,Y -659.538,Z 994.412,A 0.000,B 0.000,C 90.000,E1 290.120} C_DIS
LIN {X 0.085,Y -657.106,Z 994.411,A 0.000,B 0.000,C 90.000,E1 289.885} C_DIS
LIN {X 0.001,Y -647.672,Z 994.407,A 0.000,B 0.000,C 90.000,E1 289.322} C_DIS
LIN {X 0.018,Y -644.544,Z 994.406,A 0.000,B 0.000,C 90.000,E1 289.141} C_DIS
LIN {X -0.058,Y -641.710,Z 994.405,A 0.000,B 0.000,C 90.000,E1 288.906} C_DIS
LIN {X -0.099,Y -641.701,Z 994.405,A 0.000,B 0.000,C 90.000,E1 288.906} C_DIS
LIN {X -0.219,Y -641.669,Z 994.405,A 0.000,B 0.000,C 90.000,E1 288.852} C_DIS
LIN {X -0.072,Y -643.656,Z 994.402,A 0.000,B 0.000,C 90.000,E1 288.362} C_DIS
LIN {X 0.031,Y -652.011,Z 994.394,A 0.000,B 0.000,C 90.000,E1 286.985} C_DIS
LIN {X -0.188,Y -655.422,Z 994.391,A 0.000,B 0.000,C 90.000,E1 286.386} C_DIS
LIN {X -0.386,Y -658.228,Z 994.388,A 0.000,B 0.000,C 90.000,E1 285.788} C_DIS
LIN {X 0.107,Y -660.872,Z 994.383,A 0.000,B 0.000,C 90.000,E1 285.009} C_DIS
LIN {X -0.090,Y -662.146,Z 994.381,A 0.000,B 0.000,C 90.000,E1 284.537} C_DIS
LIN {X 0.276,Y -663.520,Z 994.377,A 0.000,B 0.000,C 90.000,E1 283.772} C_DIS
LIN {X 0.098,Y -664.148,Z 994.374,A 0.000,B 0.000,C 90.000,E1 283.300} C_DIS
LIN {X -0.163,Y -664.672,Z 994.370,A 0.000,B 0.000,C 90.000,E1 282.591} C_DIS
LIN {X 0.313,Y -664.829,Z 994.367,A 0.000,B 0.000,C 90.000,E1 282.063} C_DIS
LIN {X 0.139,Y -664.795,Z 994.365,A 0.000,B 0.000,C 90.000,E1 281.591} C_DIS
LIN {X -0.255,Y -664.305,Z 994.360,A 0.000,B 0.000,C 90.000,E1 280.894} C_DIS
LIN {X 0.215,Y -663.815,Z 994.358,A 0.000,B 0.000,C 90.000,E1 280.366} C_DIS
LIN {X -0.089,Y -662.976,Z 994.355,A 0.000,B 0.000,C 90.000,E1 279.905} C_DIS
LIN {X 0.368,Y -661.921,Z 994.352,A 0.000,B 0.000,C 90.000,E1 279.378} C_DIS
LIN {X 0.056,Y -660.518,Z 994.350,A 0.000,B 0.000,C 90.000,E1 278.916} C_DIS
LIN {X -0.259,Y -658.826,Z 994.347,A 0.000,B 0.000,C 90.000,E1 278.454} C_DIS
LIN {X 0.278,Y -657.905,Z 994.346,A 0.000,B 0.000,C 90.000,E1 278.163} C_DIS
LIN {X -0.053,Y -655.701,Z 994.343,A 0.000,B 0.000,C 90.000,E1 277.701} C_DIS
LIN {X 0.142,Y -652.282,Z 994.339,A 0.000,B 0.000,C 90.000,E1 277.068} C_DIS
LIN {X -0.222,Y -649.035,Z 994.337,A 0.000,B 0.000,C 90.000,E1 276.606} C_DIS
LIN {X -0.011,Y -644.168,Z 994.333,A 0.000,B 0.000,C 90.000,E1 275.967} C_DIS
LIN {X 0.148,Y -639.857,Z 994.330,A 0.000,B 0.000,C 90.000,E1 275.454} C_DIS
LIN {X -0.266,Y -635.076,Z 994.328,A 0.000,B 0.000,C 90.000,E1 274.992} C_DIS
LIN {X 0.020,Y -628.528,Z 994.324,A 0.000,B 0.000,C 90.000,E1 274.359} C_DIS
LIN {X 0.099,Y -621.548,Z 994.321,A 0.000,B 0.000,C 90.000,E1 273.784} C_DIS
LIN {X 0.184,Y -618.696,Z 994.320,A 0.000,B 0.000,C 90.000,E1 273.555} C_DIS
LIN {X 0.101,Y -611.060,Z 994.317,A 0.000,B 0.000,C 90.000,E1 273.037} C_DIS
LIN {X 0.278,Y -604.723,Z 994.315,A 0.000,B 0.000,C 90.000,E1 272.636} C_DIS
LIN {X 0.181,Y -598.207,Z 994.313,A 0.000,B 0.000,C 90.000,E1 272.293} C_DIS
LIN {X -0.102,Y -591.267,Z 994.311,A 0.000,B 0.000,C 90.000,E1 272.007} C_DIS
LIN {X 0.111,Y -583.946,Z 994.310,A 0.000,B 0.000,C 90.000,E1 271.718} C_DIS
LIN {X 0.256,Y -576.309,Z 994.308,A 0.000,B 0.000,C 90.000,E1 271.489} C_DIS
LIN {X 0.015,Y -570.612,Z 994.308,A 0.000,B 0.000,C 90.000,E1 271.375} C_DIS
LIN {X -0.008,Y -564.386,Z 994.307,A 0.000,B 0.000,C 90.000,E1 271.260} C_DIS
LIN {X 0.083,Y -558.084,Z 994.307,A 0.000,B 0.000,C 90.000,E1 271.203} C_DIS
LIN {X 0.039,Y -543.333,Z 994.307,A 0.000,B 0.000,C 90.000,E1 271.203} C_DIS
LIN {X 0.158,Y -542.879,Z 994.306,A 0.000,B 0.000,C 90.000,E1 271.031} C_DIS
LIN {X 0.174,Y -542.273,Z 994.303,A 0.000,B 0.000,C 90.000,E1 270.458} C_DIS
LIN {X -0.209,Y -541.086,Z 994.293,A 0.000,B 0.000,C 90.000,E1 268.797} C_DIS
LIN {X -0.086,Y -540.120,Z 994.285,A 0.000,B 0.000,C 90.000,E1 267.364} C_DIS
LIN {X 0.053,Y -539.066,Z 994.277,A 0.000,B 0.000,C 90.000,E1 265.927} C_DIS
LIN {X 0.179,Y -538.004,Z 994.270,A 0.000,B 0.000,C 90.000,E1 264.489} C_DIS
LIN {X -0.260,Y -536.727,Z 994.262,A 0.000,B 0.000,C 90.000,E1 263.109} C_DIS
LIN {X -0.059,Y -535.327,Z 994.254,A 0.000,B 0.000,C 90.000,E1 261.659} C_DIS
LIN {X 0.083,Y -533.632,Z 994.244,A 0.000,B 0.000,C 90.000,E1 259.926} C_DIS
LIN {X -0.158,Y -531.794,Z 994.235,A 0.000,B 0.000,C 90.000,E1 258.229} C_DIS
LIN {X 0.005,Y -530.497,Z 994.228,A 0.000,B 0.000,C 90.000,E1 257.061} C_DIS
LIN {X -0.219,Y -528.898,Z 994.220,A 0.000,B 0.000,C 90.000,E1 255.644} C_DIS
LIN {X 0.030,Y -526.027,Z 994.206,A 0.000,B 0.000,C 90.000,E1 253.015} C_DIS
LIN {X -0.131,Y -524.709,Z 994.199,A 0.000,B 0.000,C 90.000,E1 251.873} C_DIS
LIN {X 0.178,Y -523.293,Z 994.193,A 0.000,B 0.000,C 90.000,E1 250.678} C_DIS
LIN {X -0.039,Y -521.071,Z 994.183,A 0.000,B 0.000,C 90.000,E1 248.954} C_DIS
LIN {X 0.182,Y -518.796,Z 994.173,A 0.000,B 0.000,C 90.000,E1 247.177} C_DIS
LIN {X -0.207,Y -517.145,Z 994.167,A 0.000,B 0.000,C 90.000,E1 246.049} C_DIS
LIN {X 0.067,Y -515.413,Z 994.160,A 0.000,B 0.000,C 90.000,E1 244.845} C_DIS
LIN {X -0.145,Y -513.588,Z 994.154,A 0.000,B 0.000,C 90.000,E1 243.691} C_DIS
LIN {X 0.061,Y -510.831,Z 994.144,A 0.000,B 0.000,C 90.000,E1 241.897} C_DIS
LIN {X -0.010,Y -507.833,Z 994.134,A 0.000,B 0.000,C 90.000,E1 240.127} C_DIS
LIN {X -0.100,Y -505.661,Z 994.128,A 0.000,B 0.000,C 90.000,E1 238.948} C_DIS
LIN {X 0.031,Y -503.355,Z 994.121,A 0.000,B 0.000,C 90.000,E1 237.740} C_DIS
LIN {X -0.020,Y -500.878,Z 994.114,A 0.000,B 0.000,C 90.000,E1 236.548} C_DIS
LIN {X 0.030,Y -498.215,Z 994.108,A 0.000,B 0.000,C 90.000,E1 235.341} C_DIS
LIN {X 0.043,Y -496.148,Z 994.102,A 0.000,B 0.000,C 90.000,E1 234.436} C_DIS
LIN {X 0.178,Y -493.213,Z 994.096,A 0.000,B 0.000,C 90.000,E1 233.210} C_DIS
LIN {X 0.103,Y -488.050,Z 994.084,A 0.000,B 0.000,C 90.000,E1 231.090} C_DIS
LIN {X -0.085,Y -485.866,Z 994.079,A 0.000,B 0.000,C 90.000,E1 230.194} C_DIS
LIN {X 0.016,Y -482.365,Z 994.070,A 0.000,B 0.000,C 90.000,E1 228.647} C_DIS
LIN {X -0.103,Y -475.666,Z 994.053,A 0.000,B 0.000,C 90.000,E1 225.567} C_DIS
LIN {X -0.257,Y -472.355,Z 994.044,A 0.000,B 0.000,C 90.000,E1 224.028} C_DIS
LIN {X -0.136,Y -468.913,Z 994.036,A 0.000,B 0.000,C 90.000,E1 222.447} C_DIS
LIN {X 0.011,Y -464.767,Z 994.025,A 0.000,B 0.000,C 90.000,E1 220.539} C_DIS
LIN {X 0.119,Y -460.470,Z 994.015,A 0.000,B 0.000,C 90.000,E1 218.624} C_DIS
LIN {X 0.121,Y -456.263,Z 994.004,A 0.000,B 0.000,C 90.000,E1 216.710} C_DIS
LIN {X -0.158,Y -452.050,Z 993.993,A 0.000,B 0.000,C 90.000,E1 214.818} C_DIS
LIN {X -0.156,Y -447.843,Z 993.983,A 0.000,B 0.000,C 90.000,E1 212.880} C_DIS
LIN {X -0.184,Y -444.299,Z 993.974,A 0.000,B 0.000,C 90.000,E1 211.258} C_DIS
LIN {X -0.125,Y -440.768,Z 993.964,A 0.000,B 0.000,C 90.000,E1 209.617} C_DIS
LIN {X 0.132,Y -434.847,Z 993.950,A 0.000,B 0.000,C 90.000,E1 206.950} C_DIS
LIN {X 0.189,Y -431.112,Z 993.941,A 0.000,B 0.000,C 90.000,E1 205.283} C_DIS
LIN {X 0.147,Y -425.787,Z 993.928,A 0.000,B 0.000,C 90.000,E1 202.950} C_DIS
LIN {X -0.159,Y -421.284,Z 993.916,A 0.000,B 0.000,C 90.000,E1 200.972} C_DIS
LIN {X 0.137,Y -418.495,Z 993.909,A 0.000,B 0.000,C 90.000,E1 199.577} C_DIS
LIN {X 0.070,Y -413.179,Z 993.894,A 0.000,B 0.000,C 90.000,E1 196.858} C_DIS
LIN {X -0.148,Y -409.503,Z 993.882,A 0.000,B 0.000,C 90.000,E1 194.828} C_DIS
LIN {X 0.124,Y -406.606,Z 993.873,A 0.000,B 0.000,C 90.000,E1 193.063} C_DIS
LIN {X -0.061,Y -403.062,Z 993.861,A 0.000,B 0.000,C 90.000,E1 191.007} C_DIS
LIN {X -0.141,Y -397.927,Z 993.844,A 0.000,B 0.000,C 90.000,E1 187.871} C_DIS
LIN {X 0.157,Y -397.239,Z 993.840,A 0.000,B 0.000,C 90.000,E1 187.125} C_DIS
LIN {X 0.132,Y -396.953,Z 993.838,A 0.000,B 0.000,C 90.000,E1 186.777} C_DIS
LIN {X 0.002,Y -396.855,Z 993.832,A 0.000,B 0.000,C 90.000,E1 185.739} C_DIS
LIN {X -0.030,Y -397.072,Z 993.830,A 0.000,B 0.000,C 90.000,E1 185.391} C_DIS
LIN {X -0.099,Y -397.565,Z 993.828,A 0.000,B 0.000,C 90.000,E1 185.049} C_DIS
LIN {X -0.132,Y -398.239,Z 993.826,A 0.000,B 0.000,C 90.000,E1 184.702} C_DIS
LIN {X -0.197,Y -399.130,Z 993.824,A 0.000,B 0.000,C 90.000,E1 184.359} C_DIS
LIN {X 0.144,Y -401.021,Z 993.821,A 0.000,B 0.000,C 90.000,E1 183.784} C_DIS
LIN {X 0.118,Y -401.847,Z 993.820,A 0.000,B 0.000,C 90.000,E1 183.612} C_DIS
LIN {X 0.110,Y -406.261,Z 993.816,A 0.000,B 0.000,C 90.000,E1 182.865} C_DIS
LIN {X 0.065,Y -411.623,Z 993.812,A 0.000,B 0.000,C 90.000,E1 182.178} C_DIS
LIN {X -0.040,Y -419.954,Z 993.807,A 0.000,B 0.000,C 90.000,E1 181.260} C_DIS
LIN {X 0.079,Y -435.767,Z 993.798,A 0.000,B 0.000,C 90.000,E1 179.599} C_DIS
LIN {X -0.112,Y -444.321,Z 993.793,A 0.000,B 0.000,C 90.000,E1 178.740} C_DIS
LIN {X -0.101,Y -449.928,Z 993.790,A 0.000,B 0.000,C 90.000,E1 178.165} C_DIS
LIN {X 0.171,Y -459.580,Z 993.784,A 0.000,B 0.000,C 90.000,E1 177.078} C_DIS
LIN {X -0.031,Y -463.469,Z 993.782,A 0.000,B 0.000,C 90.000,E1 176.674} C_DIS
LIN {X -0.208,Y -470.072,Z 993.777,A 0.000,B 0.000,C 90.000,E1 175.927} C_DIS
LIN {X 0.130,Y -477.618,Z 993.772,A 0.000,B 0.000,C 90.000,E1 174.951} C_DIS
LIN {X -0.110,Y -483.644,Z 993.768,A 0.000,B 0.000,C 90.000,E1 174.204} C_DIS
LIN {X 0.060,Y -491.525,Z 993.762,A 0.000,B 0.000,C 90.000,E1 173.109} C_DIS
LIN {X -0.010,Y -499.008,Z 993.756,A 0.000,B 0.000,C 90.000,E1 172.064} C_DIS
LIN {X 0.187,Y -505.300,Z 993.751,A 0.000,B 0.000,C 90.000,E1 171.141} C_DIS
LIN {X -0.093,Y -513.309,Z 993.744,A 0.000,B 0.000,C 90.000,E1 169.982} C_DIS
LIN {X -0.173,Y -520.608,Z 993.738,A 0.000,B 0.000,C 90.000,E1 168.814} C_DIS
LIN {X 0.214,Y -525.165,Z 993.734,A 0.000,B 0.000,C 90.000,E1 168.049} C_DIS
LIN {X -0.022,Y -531.343,Z 993.728,A 0.000,B 0.000,C 90.000,E1 167.061} C_DIS
LIN {X 0.117,Y -539.055,Z 993.721,A 0.000,B 0.000,C 90.000,E1 165.755} C_DIS
LIN {X 0.169,Y -544.981,Z 993.715,A 0.000,B 0.000,C 90.000,E1 164.755} C_DIS
LIN {X -0.149,Y -555.455,Z 993.705,A 0.000,B 0.000,C 90.000,E1 162.960} C_DIS
LIN {X -0.266,Y -562.918,Z 993.698,A 0.000,B 0.000,C 90.000,E1 161.583} C_DIS
LIN {X -0.077,Y -570.175,Z 993.690,A 0.000,B 0.000,C 90.000,E1 160.188} C_DIS
LIN {X -0.011,Y -576.379,Z 993.683,A 0.000,B 0.000,C 90.000,E1 158.954} C_DIS
LIN {X -0.080,Y -579.613,Z 993.679,A 0.000,B 0.000,C 90.000,E1 158.284} C_DIS
LIN {X -0.269,Y -583.886,Z 993.674,A 0.000,B 0.000,C 90.000,E1 157.358} C_DIS
LIN {X 0.302,Y -588.626,Z 993.668,A 0.000,B 0.000,C 90.000,E1 156.230} C_DIS
LIN {X -0.277,Y -591.838,Z 993.664,A 0.000,B 0.000,C 90.000,E1 155.485} C_DIS
LIN {X 0.053,Y -593.831,Z 993.661,A 0.000,B 0.000,C 90.000,E1 154.921} C_DIS
LIN {X -0.316,Y -597.607,Z 993.655,A 0.000,B 0.000,C 90.000,E1 153.896} C_DIS
LIN {X -0.101,Y -601.002,Z 993.649,A 0.000,B 0.000,C 90.000,E1 152.820} C_DIS
LIN {X -0.033,Y -603.452,Z 993.645,A 0.000,B 0.000,C 90.000,E1 152.025} C_DIS
LIN {X -0.096,Y -608.041,Z 993.636,A 0.000,B 0.000,C 90.000,E1 150.461} C_DIS
LIN {X 0.009,Y -611.094,Z 993.630,A 0.000,B 0.000,C 90.000,E1 149.410} C_DIS
LIN {X -0.092,Y -614.761,Z 993.623,A 0.000,B 0.000,C 90.000,E1 148.122} C_DIS
LIN {X -0.126,Y -618.364,Z 993.616,A 0.000,B 0.000,C 90.000,E1 146.834} C_DIS
LIN {X 0.003,Y -624.160,Z 993.604,A 0.000,B 0.000,C 90.000,E1 144.769} C_DIS
LIN {X -0.199,Y -628.499,Z 993.596,A 0.000,B 0.000,C 90.000,E1 143.256} C_DIS
LIN {X 0.061,Y -633.448,Z 993.586,A 0.000,B 0.000,C 90.000,E1 141.457} C_DIS
LIN {X 0.171,Y -636.252,Z 993.580,A 0.000,B 0.000,C 90.000,E1 140.436} C_DIS
LIN {X 0.211,Y -639.700,Z 993.573,A 0.000,B 0.000,C 90.000,E1 139.175} C_DIS
LIN {X 0.248,Y -643.096,Z 993.566,A 0.000,B 0.000,C 90.000,E1 137.919} C_DIS
LIN {X -0.347,Y -649.384,Z 993.554,A 0.000,B 0.000,C 90.000,E1 135.729} C_DIS
LIN {X 0.146,Y -656.321,Z 993.542,A 0.000,B 0.000,C 90.000,E1 133.461} C_DIS
LIN {X 0.000,Y -661.295,Z 993.533,A 0.000,B 0.000,C 90.000,E1 132.000} C_DIS
LIN {X -0.034,Y -665.565,Z 993.527,A 0.000,B 0.000,C 90.000,E1 130.782} C_DIS
LIN {X -0.008,Y -670.567,Z 993.518,A 0.000,B 0.000,C 90.000,E1 129.322} C_DIS
LIN {X -0.338,Y -673.615,Z 993.513,A 0.000,B 0.000,C 90.000,E1 128.382} C_DIS
LIN {X 0.064,Y -678.703,Z 993.504,A 0.000,B 0.000,C 90.000,E1 126.664} C_DIS
LIN {X 0.189,Y -683.464,Z 993.494,A 0.000,B 0.000,C 90.000,E1 124.978} C_DIS
LIN {X 0.013,Y -686.143,Z 993.489,A 0.000,B 0.000,C 90.000,E1 124.040} C_DIS
LIN {X -0.110,Y -689.779,Z 993.481,A 0.000,B 0.000,C 90.000,E1 122.625} C_DIS
LIN {X -0.149,Y -693.490,Z 993.473,A 0.000,B 0.000,C 90.000,E1 121.209} C_DIS
LIN {X -0.023,Y -695.749,Z 993.468,A 0.000,B 0.000,C 90.000,E1 120.256} C_DIS
LIN {X -0.226,Y -697.571,Z 993.463,A 0.000,B 0.000,C 90.000,E1 119.333} C_DIS
LIN {X 0.293,Y -698.402,Z 993.460,A 0.000,B 0.000,C 90.000,E1 118.821} C_DIS
LIN {X -0.145,Y -699.325,Z 993.456,A 0.000,B 0.000,C 90.000,E1 118.153} C_DIS
LIN {X 0.390,Y -699.860,Z 993.454,A 0.000,B 0.000,C 90.000,E1 117.641} C_DIS
LIN {X 0.098,Y -701.256,Z 993.445,A 0.000,B 0.000,C 90.000,E1 116.027} C_DIS
LIN {X -0.014,Y -701.821,Z 993.441,A 0.000,B 0.000,C 90.000,E1 115.335} C_DIS
LIN {X 0.145,Y -702.125,Z 993.434,A 0.000,B 0.000,C 90.000,E1 114.155} C_DIS
LIN {X 0.055,Y -701.638,Z 993.432,A 0.000,B 0.000,C 90.000,E1 113.695} C_DIS
LIN {X 0.048,Y -701.179,Z 993.430,A 0.000,B 0.000,C 90.000,E1 113.462} C_DIS
LIN {X -0.195,Y -698.480,Z 993.427,A 0.000,B 0.000,C 90.000,E1 112.898} C_DIS
LIN {X -0.063,Y -697.610,Z 993.427,A 0.000,B 0.000,C 90.000,E1 112.770} C_DIS
LIN {X 0.195,Y -695.040,Z 993.425,A 0.000,B 0.000,C 90.000,E1 112.514} C_DIS
LIN {X -0.291,Y -692.445,Z 993.424,A 0.000,B 0.000,C 90.000,E1 112.333} C_DIS
LIN {X -0.061,Y -690.956,Z 993.423,A 0.000,B 0.000,C 90.000,E1 112.206} C_DIS
LIN {X 0.167,Y -688.464,Z 993.423,A 0.000,B 0.000,C 90.000,E1 112.078} C_DIS
LIN {X -0.010,Y -684.367,Z 993.422,A 0.000,B 0.000,C 90.000,E1 111.950} C_DIS
LIN {X 0.177,Y -676.166,Z 993.421,A 0.000,B 0.000,C 90.000,E1 111.791} C_DIS
LIN {X 0.219,Y -673.459,Z 993.421,A 0.000,B 0.000,C 90.000,E1 111.770} C_DIS
LIN {X 0.162,Y -620.176,Z 993.421,A 0.000,B 0.000,C 90.000,E1 111.770} C_DIS
LIN {X -0.106,Y -616.483,Z 993.421,A 0.000,B 0.000,C 90.000,E1 111.716} C_DIS
LIN {X -0.350,Y -609.551,Z 993.419,A 0.000,B 0.000,C 90.000,E1 111.535} C_DIS
LIN {X -0.229,Y -602.288,Z 993.418,A 0.000,B 0.000,C 90.000,E1 111.227} C_DIS
LIN {X 0.022,Y -596.170,Z 993.416,A 0.000,B 0.000,C 90.000,E1 110.865} C_DIS
LIN {X 0.145,Y -589.934,Z 993.414,A 0.000,B 0.000,C 90.000,E1 110.429} C_DIS
LIN {X 0.319,Y -577.772,Z 993.408,A 0.000,B 0.000,C 90.000,E1 109.450} C_DIS
LIN {X 0.130,Y -573.570,Z 993.406,A 0.000,B 0.000,C 90.000,E1 109.141} C_DIS
LIN {X -0.138,Y -565.469,Z 993.404,A 0.000,B 0.000,C 90.000,E1 108.671} C_DIS
LIN {X 0.231,Y -553.803,Z 993.401,A 0.000,B 0.000,C 90.000,E1 108.055} C_DIS
LIN {X 0.079,Y -551.311,Z 993.400,A 0.000,B 0.000,C 90.000,E1 107.946} C_DIS
LIN {X -0.020,Y -550.315,Z 993.399,A 0.000,B 0.000,C 90.000,E1 107.873} C_DIS
LIN {X -0.200,Y -549.151,Z 993.399,A 0.000,B 0.000,C 90.000,E1 107.764} C_DIS
LIN {X -0.241,Y -549.139,Z 993.399,A 0.000,B 0.000,C 90.000,E1 107.764} C_DIS
LIN {X 0.016,Y -548.699,Z 993.397,A 0.000,B 0.000,C 90.000,E1 107.457} C_DIS
LIN {X 0.223,Y -548.807,Z 993.393,A 0.000,B 0.000,C 90.000,E1 106.732} C_DIS
LIN {X 0.233,Y -549.313,Z 993.387,A 0.000,B 0.000,C 90.000,E1 105.607} C_DIS
LIN {X 0.286,Y -550.464,Z 993.374,A 0.000,B 0.000,C 90.000,E1 103.355} C_DIS
LIN {X 0.177,Y -553.634,Z 993.354,A 0.000,B 0.000,C 90.000,E1 99.726} C_DIS
LIN {X 0.073,Y -555.125,Z 993.346,A 0.000,B 0.000,C 90.000,E1 98.341} C_DIS
LIN {X 0.076,Y -556.615,Z 993.339,A 0.000,B 0.000,C 90.000,E1 96.947} C_DIS
LIN {X -0.101,Y -557.666,Z 993.333,A 0.000,B 0.000,C 90.000,E1 95.853} C_DIS
LIN {X -0.189,Y -558.658,Z 993.325,A 0.000,B 0.000,C 90.000,E1 94.473} C_DIS
LIN {X 0.178,Y -559.346,Z 993.319,A 0.000,B 0.000,C 90.000,E1 93.326} C_DIS
LIN {X 0.092,Y -560.097,Z 993.311,A 0.000,B 0.000,C 90.000,E1 91.949} C_DIS
LIN {X 0.108,Y -560.924,Z 993.302,A 0.000,B 0.000,C 90.000,E1 90.286} C_DIS
LIN {X 0.031,Y -561.570,Z 993.294,A 0.000,B 0.000,C 90.000,E1 88.912} C_DIS
LIN {X -0.024,Y -561.893,Z 993.286,A 0.000,B 0.000,C 90.000,E1 87.535} C_DIS
LIN {X 0.152,Y -562.212,Z 993.276,A 0.000,B 0.000,C 90.000,E1 85.584} C_DIS
LIN {X -0.038,Y -562.519,Z 993.263,A 0.000,B 0.000,C 90.000,E1 83.394} C_DIS
LIN {X 0.252,Y -562.912,Z 993.253,A 0.000,B 0.000,C 90.000,E1 81.432} C_DIS
LIN {X -0.229,Y -563.654,Z 993.240,A 0.000,B 0.000,C 90.000,E1 79.275} C_DIS
LIN {X -0.076,Y -564.272,Z 993.233,A 0.000,B 0.000,C 90.000,E1 77.881} C_DIS
LIN {X 0.155,Y -564.896,Z 993.227,A 0.000,B 0.000,C 90.000,E1 76.756} C_DIS
LIN {X 0.139,Y -566.518,Z 993.213,A 0.000,B 0.000,C 90.000,E1 74.283} C_DIS
LIN {X 0.130,Y -567.907,Z 993.202,A 0.000,B 0.000,C 90.000,E1 72.362} C_DIS
LIN {X -0.343,Y -568.874,Z 993.195,A 0.000,B 0.000,C 90.000,E1 71.040} C_DIS
LIN {X -0.083,Y -569.715,Z 993.187,A 0.000,B 0.000,C 90.000,E1 69.645} C_DIS
LIN {X 0.040,Y -570.354,Z 993.181,A 0.000,B 0.000,C 90.000,E1 68.539} C_DIS
LIN {X -0.179,Y -571.163,Z 993.172,A 0.000,B 0.000,C 90.000,E1 66.922} C_DIS
LIN {X 0.189,Y -571.605,Z 993.166,A 0.000,B 0.000,C 90.000,E1 65.793} C_DIS
LIN {X 0.045,Y -572.058,Z 993.160,A 0.000,B 0.000,C 90.000,E1 64.717} C_DIS
LIN {X 0.089,Y -572.567,Z 993.151,A 0.000,B 0.000,C 90.000,E1 63.076} C_DIS
LIN {X 0.154,Y -572.961,Z 993.141,A 0.000,B 0.000,C 90.000,E1 61.435} C_DIS
LIN {X 0.116,Y -573.295,Z 993.134,A 0.000,B 0.000,C 90.000,E1 60.078} C_DIS
LIN {X -0.004,Y -573.539,Z 993.125,A 0.000,B 0.000,C 90.000,E1 58.456} C_DIS
LIN {X -0.111,Y -573.745,Z 993.116,A 0.000,B 0.000,C 90.000,E1 56.834} C_DIS
LIN {X -0.048,Y -573.861,Z 993.108,A 0.000,B 0.000,C 90.000,E1 55.468} C_DIS
LIN {X 0.050,Y -573.843,Z 993.104,A 0.000,B 0.000,C 90.000,E1 54.642} C_DIS
LIN {X 0.162,Y -573.679,Z 993.098,A 0.000,B 0.000,C 90.000,E1 53.543} C_DIS
LIN {X -0.063,Y -573.294,Z 993.092,A 0.000,B 0.000,C 90.000,E1 52.477} C_DIS
LIN {X 0.056,Y -572.737,Z 993.086,A 0.000,B 0.000,C 90.000,E1 51.376} C_DIS
LIN {X 0.167,Y -572.042,Z 993.079,A 0.000,B 0.000,C 90.000,E1 50.275} C_DIS
LIN {X -0.173,Y -571.098,Z 993.073,A 0.000,B 0.000,C 90.000,E1 49.218} C_DIS
LIN {X -0.223,Y -570.285,Z 993.069,A 0.000,B 0.000,C 90.000,E1 48.405} C_DIS
LIN {X 0.093,Y -569.321,Z 993.064,A 0.000,B 0.000,C 90.000,E1 47.553} C_DIS
LIN {X -0.015,Y -568.167,Z 993.060,A 0.000,B 0.000,C 90.000,E1 46.743} C_DIS
LIN {X -0.032,Y -566.375,Z 993.054,A 0.000,B 0.000,C 90.000,E1 45.648} C_DIS
LIN {X 0.318,Y -564.185,Z 993.048,A 0.000,B 0.000,C 90.000,E1 44.514} C_DIS
LIN {X 0.158,Y -562.299,Z 993.043,A 0.000,B 0.000,C 90.000,E1 43.704} C_DIS
LIN {X -0.081,Y -560.926,Z 993.040,A 0.000,B 0.000,C 90.000,E1 43.176} C_DIS
LIN {X -0.198,Y -557.766,Z 993.034,A 0.000,B 0.000,C 90.000,E1 42.081} C_DIS
LIN {X -0.017,Y -555.063,Z 993.029,A 0.000,B 0.000,C 90.000,E1 41.229} C_DIS
LIN {X 0.129,Y -552.057,Z 993.024,A 0.000,B 0.000,C 90.000,E1 40.378} C_DIS
LIN {X -0.171,Y -549.820,Z 993.021,A 0.000,B 0.000,C 90.000,E1 39.850} C_DIS
LIN {X 0.134,Y -546.780,Z 993.017,A 0.000,B 0.000,C 90.000,E1 39.116} C_DIS
LIN {X -0.170,Y -542.834,Z 993.013,A 0.000,B 0.000,C 90.000,E1 38.302} C_DIS
LIN {X 0.083,Y -537.964,Z 993.007,A 0.000,B 0.000,C 90.000,E1 37.282} C_DIS
LIN {X -0.210,Y -531.953,Z 993.001,A 0.000,B 0.000,C 90.000,E1 36.171} C_DIS
LIN {X -0.083,Y -527.955,Z 992.997,A 0.000,B 0.000,C 90.000,E1 35.438} C_DIS
LIN {X 0.295,Y -524.542,Z 992.994,A 0.000,B 0.000,C 90.000,E1 34.818} C_DIS
LIN {X -0.007,Y -518.190,Z 992.988,A 0.000,B 0.000,C 90.000,E1 33.833} C_DIS
LIN {X 0.010,Y -514.382,Z 992.985,A 0.000,B 0.000,C 90.000,E1 33.245} C_DIS
LIN {X 0.035,Y -511.382,Z 992.982,A 0.000,B 0.000,C 90.000,E1 32.801} C_DIS
LIN {X -0.026,Y -506.039,Z 992.978,A 0.000,B 0.000,C 90.000,E1 32.084} C_DIS
LIN {X -0.013,Y -500.131,Z 992.974,A 0.000,B 0.000,C 90.000,E1 31.337} C_DIS
LIN {X 0.088,Y -496.379,Z 992.972,A 0.000,B 0.000,C 90.000,E1 30.875} C_DIS
LIN {X -0.251,Y -492.377,Z 992.969,A 0.000,B 0.000,C 90.000,E1 30.463} C_DIS
LIN {X -0.229,Y -486.882,Z 992.966,A 0.000,B 0.000,C 90.000,E1 29.873} C_DIS
LIN {X -0.088,Y -476.985,Z 992.960,A 0.000,B 0.000,C 90.000,E1 28.871} C_DIS
LIN {X -0.015,Y -471.208,Z 992.957,A 0.000,B 0.000,C 90.000,E1 28.309} C_DIS
LIN {X -0.230,Y -460.887,Z 992.952,A 0.000,B 0.000,C 90.000,E1 27.385} C_DIS
LIN {X -0.066,Y -450.254,Z 992.947,A 0.000,B 0.000,C 90.000,E1 26.437} C_DIS
LIN {X -0.164,Y -432.188,Z 992.938,A 0.000,B 0.000,C 90.000,E1 24.899} C_DIS
LIN {X -0.166,Y -417.308,Z 992.931,A 0.000,B 0.000,C 90.000,E1 23.515} C_DIS
LIN {X -0.050,Y -404.131,Z 992.923,A 0.000,B 0.000,C 90.000,E1 22.153} C_DIS
LIN {X -0.038,Y -398.643,Z 992.920,A 0.000,B 0.000,C 90.000,E1 21.535} C_DIS
LIN {X -0.155,Y -395.154,Z 992.917,A 0.000,B 0.000,C 90.000,E1 21.099} C_DIS
LIN {X -0.056,Y -392.247,Z 992.914,A 0.000,B 0.000,C 90.000,E1 20.556} C_DIS
LIN {X -0.126,Y -390.851,Z 992.912,A 0.000,B 0.000,C 90.000,E1 20.120} C_DIS
LIN {X 0.203,Y -390.140,Z 992.908,A 0.000,B 0.000,C 90.000,E1 19.450} C_DIS
LIN {X -0.082,Y -390.304,Z 992.904,A 0.000,B 0.000,C 90.000,E1 18.779} C_DIS
LIN {X 0.205,Y -394.140,Z 992.883,A 0.000,B 0.000,C 90.000,E1 14.828} C_DIS
LIN {X 0.183,Y -399.245,Z 992.861,A 0.000,B 0.000,C 90.000,E1 10.950} C_DIS
LIN {X 0.048,Y -405.793,Z 992.840,A 0.000,B 0.000,C 90.000,E1 7.125} C_DIS
LIN {X 0.027,Y -411.371,Z 992.824,A 0.000,B 0.000,C 90.000,E1 4.359} C_DIS
LIN {X 0.065,Y -415.144,Z 992.815,A 0.000,B 0.000,C 90.000,E1 2.636} C_DIS
LIN {X 0.116,Y -417.374,Z 992.809,A 0.000,B 0.000,C 90.000,E1 1.604} C_DIS
LIN {X 0.135,Y -418.296,Z 992.807,A 0.000,B 0.000,C 90.000,E1 1.260} C_DIS
LIN {X 0.157,Y -419.461,Z 992.805,A 0.000,B 0.000,C 90.000,E1 0.917} C_DIS
LIN {X 0.110,Y -423.438,Z 992.801,A 0.000,B 0.000,C 90.000,E1 0.115} C_DIS
LIN {X 0.161,Y -426.604,Z 992.799,A 0.000,B 0.000,C 90.000,E1 359.771} C_DIS
LIN {X -0.206,Y -428.713,Z 992.798,A 0.000,B 0.000,C 90.000,E1 359.599} C_DIS
LIN {X -0.028,Y -434.292,Z 992.796,A 0.000,B 0.000,C 90.000,E1 359.198} C_DIS
LIN {X -0.111,Y -448.941,Z 992.791,A 0.000,B 0.000,C 90.000,E1 358.396} C_DIS
LIN {X -0.050,Y -464.083,Z 992.786,A 0.000,B 0.000,C 90.000,E1 357.535} C_DIS
LIN {X 0.037,Y -484.193,Z 992.780,A 0.000,B 0.000,C 90.000,E1 356.388} C_DIS
LIN {X -0.081,Y -497.303,Z 992.776,A 0.000,B 0.000,C 90.000,E1 355.641} C_DIS
LIN {X -0.036,Y -508.384,Z 992.772,A 0.000,B 0.000,C 90.000,E1 354.951} C_DIS
LIN {X 0.019,Y -517.777,Z 992.768,A 0.000,B 0.000,C 90.000,E1 354.318} C_DIS
LIN {X -0.237,Y -526.842,Z 992.765,A 0.000,B 0.000,C 90.000,E1 353.685} C_DIS
LIN {X -0.226,Y -534.163,Z 992.762,A 0.000,B 0.000,C 90.000,E1 353.109} C_DIS
LIN {X 0.065,Y -541.109,Z 992.758,A 0.000,B 0.000,C 90.000,E1 352.470} C_DIS
LIN {X -0.097,Y -547.760,Z 992.755,A 0.000,B 0.000,C 90.000,E1 351.837} C_DIS
LIN {X -0.180,Y -552.943,Z 992.752,A 0.000,B 0.000,C 90.000,E1 351.310} C_DIS
LIN {X 0.047,Y -557.794,Z 992.749,A 0.000,B 0.000,C 90.000,E1 350.735} C_DIS
LIN {X 0.078,Y -563.294,Z 992.745,A 0.000,B 0.000,C 90.000,E1 350.038} C_DIS
LIN {X 0.239,Y -568.201,Z 992.741,A 0.000,B 0.000,C 90.000,E1 349.342} C_DIS
LIN {X 0.041,Y -571.777,Z 992.738,A 0.000,B 0.000,C 90.000,E1 348.814} C_DIS
LIN {X -0.166,Y -577.479,Z 992.733,A 0.000,B 0.000,C 90.000,E1 347.881} C_DIS
LIN {X 0.146,Y -583.270,Z 992.727,A 0.000,B 0.000,C 90.000,E1 346.769} C_DIS
LIN {X 0.199,Y -588.062,Z 992.721,A 0.000,B 0.000,C 90.000,E1 345.825} C_DIS
LIN {X 0.234,Y -593.244,Z 992.715,A 0.000,B 0.000,C 90.000,E1 344.755} C_DIS
LIN {X 0.063,Y -596.928,Z 992.711,A 0.000,B 0.000,C 90.000,E1 343.976} C_DIS
LIN {X -0.070,Y -600.480,Z 992.707,A 0.000,B 0.000,C 90.000,E1 343.196} C_DIS
LIN {X 0.125,Y -604.857,Z 992.701,A 0.000,B 0.000,C 90.000,E1 342.127} C_DIS
LIN {X -0.012,Y -609.141,Z 992.695,A 0.000,B 0.000,C 90.000,E1 341.094} C_DIS
LIN {X -0.089,Y -613.081,Z 992.689,A 0.000,B 0.000,C 90.000,E1 340.061} C_DIS
LIN {X 0.138,Y -615.784,Z 992.685,A 0.000,B 0.000,C 90.000,E1 339.263} C_DIS
LIN {X 0.123,Y -619.949,Z 992.678,A 0.000,B 0.000,C 90.000,E1 337.975} C_DIS
LIN {X -0.161,Y -623.833,Z 992.671,A 0.000,B 0.000,C 90.000,E1 336.719} C_DIS
LIN {X 0.183,Y -626.706,Z 992.665,A 0.000,B 0.000,C 90.000,E1 335.665} C_DIS
LIN {X -0.013,Y -629.395,Z 992.659,A 0.000,B 0.000,C 90.000,E1 334.665} C_DIS
LIN {X 0.093,Y -631.863,Z 992.654,A 0.000,B 0.000,C 90.000,E1 333.640} C_DIS
LIN {X 0.198,Y -633.520,Z 992.649,A 0.000,B 0.000,C 90.000,E1 332.871} C_DIS
LIN {X -0.114,Y -636.575,Z 992.641,A 0.000,B 0.000,C 90.000,E1 331.385} C_DIS
LIN {X -0.166,Y -638.452,Z 992.635,A 0.000,B 0.000,C 90.000,E1 330.383} C_DIS
LIN {X 0.367,Y -640.228,Z 992.630,A 0.000,B 0.000,C 90.000,E1 329.331} C_DIS
LIN {X 0.370,Y -641.819,Z 992.624,A 0.000,B 0.000,C 90.000,E1 328.329} C_DIS
LIN {X -0.098,Y -643.507,Z 992.617,A 0.000,B 0.000,C 90.000,E1 327.120} C_DIS
LIN {X 0.289,Y -644.696,Z 992.612,A 0.000,B 0.000,C 90.000,E1 326.087} C_DIS
LIN {X 0.161,Y -645.635,Z 992.606,A 0.000,B 0.000,C 90.000,E1 325.102} C_DIS
LIN {X 0.092,Y -646.609,Z 992.599,A 0.000,B 0.000,C 90.000,E1 323.863} C_DIS
LIN {X -0.108,Y -647.339,Z 992.592,A 0.000,B 0.000,C 90.000,E1 322.637} C_DIS
LIN {X 0.186,Y -647.748,Z 992.587,A 0.000,B 0.000,C 90.000,E1 321.618} C_DIS
LIN {X -0.075,Y -648.370,Z 992.579,A 0.000,B 0.000,C 90.000,E1 320.150} C_DIS
LIN {X -0.153,Y -649.562,Z 992.565,A 0.000,B 0.000,C 90.000,E1 317.676} C_DIS
LIN {X 0.002,Y -650.614,Z 992.557,A 0.000,B 0.000,C 90.000,E1 316.176} C_DIS
LIN {X 0.027,Y -652.083,Z 992.544,A 0.000,B 0.000,C 90.000,E1 313.947} C_DIS
LIN {X 0.270,Y -653.101,Z 992.537,A 0.000,B 0.000,C 90.000,E1 312.690} C_DIS
LIN {X -0.352,Y -653.781,Z 992.532,A 0.000,B 0.000,C 90.000,E1 311.757} C_DIS
LIN {X -0.072,Y -654.690,Z 992.524,A 0.000,B 0.000,C 90.000,E1 310.253} C_DIS
LIN {X 0.224,Y -655.417,Z 992.515,A 0.000,B 0.000,C 90.000,E1 308.749} C_DIS
LIN {X 0.113,Y -656.031,Z 992.507,A 0.000,B 0.000,C 90.000,E1 307.282} C_DIS
LIN {X -0.325,Y -656.350,Z 992.500,A 0.000,B 0.000,C 90.000,E1 306.091} C_DIS
LIN {X 0.164,Y -656.520,Z 992.494,A 0.000,B 0.000,C 90.000,E1 304.818} C_DIS
LIN {X -0.167,Y -656.845,Z 992.485,A 0.000,B 0.000,C 90.000,E1 303.372} C_DIS
LIN {X -0.078,Y -663.041,Z 992.449,A 0.000,B 0.000,C 90.000,E1 296.744} C_DIS
LIN {X -0.104,Y -665.338,Z 992.440,A 0.000,B 0.000,C 90.000,E1 295.283} C_DIS
LIN {X -0.240,Y -667.143,Z 992.434,A 0.000,B 0.000,C 90.000,E1 294.079} C_DIS
LIN {X 0.102,Y -668.379,Z 992.428,A 0.000,B 0.000,C 90.000,E1 293.078} C_DIS
LIN {X 0.150,Y -668.825,Z 992.426,A 0.000,B 0.000,C 90.000,E1 292.589} C_DIS
LIN {X -0.263,Y -668.995,Z 992.422,A 0.000,B 0.000,C 90.000,E1 291.897} C_DIS
LIN {X -0.208,Y -668.421,Z 992.419,A 0.000,B 0.000,C 90.000,E1 291.408} C_DIS
LIN {X -0.060,Y -667.976,Z 992.418,A 0.000,B 0.000,C 90.000,E1 291.153} C_DIS
LIN {X -0.177,Y -664.947,Z 992.414,A 0.000,B 0.000,C 90.000,E1 290.556} C_DIS
LIN {X -0.108,Y -664.063,Z 992.414,A 0.000,B 0.000,C 90.000,E1 290.429} C_DIS
LIN {X -0.043,Y -662.734,Z 992.413,A 0.000,B 0.000,C 90.000,E1 290.301} C_DIS
LIN {X 0.078,Y -659.655,Z 992.412,A 0.000,B 0.000,C 90.000,E1 290.066} C_DIS
LIN {X 0.324,Y -656.755,Z 992.410,A 0.000,B 0.000,C 90.000,E1 289.812} C_DIS
LIN {X 0.287,Y -645.546,Z 992.407,A 0.000,B 0.000,C 90.000,E1 289.141} C_DIS
LIN {X -0.126,Y -644.300,Z 992.406,A 0.000,B 0.000,C 90.000,E1 289.087} C_DIS
LIN {X -0.155,Y -642.904,Z 992.405,A 0.000,B 0.000,C 90.000,E1 288.960} C_DIS
LIN {X -0.196,Y -642.867,Z 992.405,A 0.000,B 0.000,C 90.000,E1 288.960} C_DIS
LIN {X 0.197,Y -642.816,Z 992.405,A 0.000,B 0.000,C 90.000,E1 288.852} C_DIS
LIN {X 0.143,Y -644.255,Z 992.403,A 0.000,B 0.000,C 90.000,E1 288.489} C_DIS
LIN {X 0.187,Y -645.616,Z 992.401,A 0.000,B 0.000,C 90.000,E1 288.236} C_DIS
LIN {X -0.331,Y -653.242,Z 992.395,A 0.000,B 0.000,C 90.000,E1 287.040} C_DIS
LIN {X 0.086,Y -656.616,Z 992.391,A 0.000,B 0.000,C 90.000,E1 286.386} C_DIS
LIN {X -0.100,Y -659.413,Z 992.388,A 0.000,B 0.000,C 90.000,E1 285.788} C_DIS
LIN {X -0.133,Y -661.247,Z 992.385,A 0.000,B 0.000,C 90.000,E1 285.300} C_DIS
LIN {X -0.234,Y -662.050,Z 992.384,A 0.000,B 0.000,C 90.000,E1 285.064} C_DIS
LIN {X 0.217,Y -663.316,Z 992.381,A 0.000,B 0.000,C 90.000,E1 284.537} C_DIS
LIN {X -0.051,Y -664.692,Z 992.377,A 0.000,B 0.000,C 90.000,E1 283.828} C_DIS
LIN {X -0.307,Y -665.549,Z 992.373,A 0.000,B 0.000,C 90.000,E1 283.119} C_DIS
LIN {X 0.175,Y -665.890,Z 992.370,A 0.000,B 0.000,C 90.000,E1 282.591} C_DIS
LIN {X 0.010,Y -666.059,Z 992.367,A 0.000,B 0.000,C 90.000,E1 282.119} C_DIS
LIN {X -0.293,Y -666.024,Z 992.365,A 0.000,B 0.000,C 90.000,E1 281.658} C_DIS
LIN {X 0.110,Y -665.589,Z 992.361,A 0.000,B 0.000,C 90.000,E1 280.894} C_DIS
LIN {X -0.065,Y -665.115,Z 992.358,A 0.000,B 0.000,C 90.000,E1 280.423} C_DIS
LIN {X 0.293,Y -664.294,Z 992.355,A 0.000,B 0.000,C 90.000,E1 279.905} C_DIS
LIN {X -0.004,Y -663.246,Z 992.353,A 0.000,B 0.000,C 90.000,E1 279.443} C_DIS
LIN {X -0.199,Y -661.888,Z 992.350,A 0.000,B 0.000,C 90.000,E1 278.973} C_DIS
LIN {X 0.250,Y -661.158,Z 992.348,A 0.000,B 0.000,C 90.000,E1 278.690} C_DIS
LIN {X 0.036,Y -659.373,Z 992.346,A 0.000,B 0.000,C 90.000,E1 278.219} C_DIS
LIN {X 0.261,Y -656.620,Z 992.342,A 0.000,B 0.000,C 90.000,E1 277.587} C_DIS
LIN {X -0.077,Y -653.920,Z 992.340,A 0.000,B 0.000,C 90.000,E1 277.125} C_DIS
LIN {X 0.179,Y -649.866,Z 992.336,A 0.000,B 0.000,C 90.000,E1 276.486} C_DIS
LIN {X -0.205,Y -646.040,Z 992.333,A 0.000,B 0.000,C 90.000,E1 276.024} C_DIS
LIN {X -0.093,Y -640.664,Z 992.330,A 0.000,B 0.000,C 90.000,E1 275.391} C_DIS
LIN {X 0.056,Y -635.857,Z 992.327,A 0.000,B 0.000,C 90.000,E1 274.878} C_DIS
LIN {X 0.072,Y -631.029,Z 992.325,A 0.000,B 0.000,C 90.000,E1 274.416} C_DIS
LIN {X 0.000,Y -624.157,Z 992.321,A 0.000,B 0.000,C 90.000,E1 273.841} C_DIS
LIN {X 0.166,Y -618.400,Z 992.319,A 0.000,B 0.000,C 90.000,E1 273.383} C_DIS
LIN {X -0.057,Y -612.230,Z 992.317,A 0.000,B 0.000,C 90.000,E1 272.980} C_DIS
LIN {X 0.275,Y -604.289,Z 992.314,A 0.000,B 0.000,C 90.000,E1 272.465} C_DIS
LIN {X 0.175,Y -597.622,Z 992.312,A 0.000,B 0.000,C 90.000,E1 272.121} C_DIS
LIN {X -0.051,Y -590.599,Z 992.310,A 0.000,B 0.000,C 90.000,E1 271.835} C_DIS
LIN {X 0.233,Y -585.188,Z 992.309,A 0.000,B 0.000,C 90.000,E1 271.604} C_DIS
LIN {X 0.217,Y -577.546,Z 992.308,A 0.000,B 0.000,C 90.000,E1 271.375} C_DIS
LIN {X -0.158,Y -571.523,Z 992.307,A 0.000,B 0.000,C 90.000,E1 271.260} C_DIS
LIN {X -0.181,Y -565.548,Z 992.306,A 0.000,B 0.000,C 90.000,E1 271.146} C_DIS
LIN {X 0.252,Y -558.280,Z 992.306,A 0.000,B 0.000,C 90.000,E1 271.031} C_DIS
LIN {X 0.206,Y -557.640,Z 992.306,A 0.000,B 0.000,C 90.000,E1 271.031} C_DIS
LIN {X 0.157,Y -543.058,Z 992.306,A 0.000,B 0.000,C 90.000,E1 271.031} C_DIS
LIN {X -0.049,Y -542.348,Z 992.303,A 0.000,B 0.000,C 90.000,E1 270.458} C_DIS
LIN {X 0.111,Y -541.172,Z 992.293,A 0.000,B 0.000,C 90.000,E1 268.740} C_DIS
LIN {X 0.235,Y -540.220,Z 992.285,A 0.000,B 0.000,C 90.000,E1 267.306} C_DIS
LIN {X -0.145,Y -538.765,Z 992.274,A 0.000,B 0.000,C 90.000,E1 265.355} C_DIS
LIN {X -0.034,Y -537.830,Z 992.268,A 0.000,B 0.000,C 90.000,E1 264.204} C_DIS
LIN {X 0.061,Y -536.824,Z 992.261,A 0.000,B 0.000,C 90.000,E1 263.053} C_DIS
LIN {X 0.206,Y -535.756,Z 992.255,A 0.000,B 0.000,C 90.000,E1 261.894} C_DIS
LIN {X -0.124,Y -533.726,Z 992.244,A 0.000,B 0.000,C 90.000,E1 259.926} C_DIS
LIN {X 0.158,Y -531.901,Z 992.234,A 0.000,B 0.000,C 90.000,E1 258.173} C_DIS
LIN {X -0.198,Y -530.600,Z 992.228,A 0.000,B 0.000,C 90.000,E1 257.061} C_DIS
LIN {X 0.094,Y -528.960,Z 992.220,A 0.000,B 0.000,C 90.000,E1 255.589} C_DIS
LIN {X -0.167,Y -526.108,Z 992.206,A 0.000,B 0.000,C 90.000,E1 253.015} C_DIS
LIN {X 0.172,Y -524.784,Z 992.199,A 0.000,B 0.000,C 90.000,E1 251.819} C_DIS
LIN {X -0.015,Y -523.368,Z 992.193,A 0.000,B 0.000,C 90.000,E1 250.678} C_DIS
LIN {X 0.256,Y -521.144,Z 992.183,A 0.000,B 0.000,C 90.000,E1 248.901} C_DIS
LIN {X -0.153,Y -519.251,Z 992.175,A 0.000,B 0.000,C 90.000,E1 247.486} C_DIS
LIN {X -0.059,Y -517.675,Z 992.168,A 0.000,B 0.000,C 90.000,E1 246.305} C_DIS
LIN {X -0.119,Y -515.497,Z 992.160,A 0.000,B 0.000,C 90.000,E1 244.845} C_DIS
LIN {X 0.132,Y -513.635,Z 992.154,A 0.000,B 0.000,C 90.000,E1 243.640} C_DIS
LIN {X -0.120,Y -510.878,Z 992.144,A 0.000,B 0.000,C 90.000,E1 241.897} C_DIS
LIN {X -0.189,Y -507.902,Z 992.134,A 0.000,B 0.000,C 90.000,E1 240.127} C_DIS
LIN {X 0.040,Y -505.159,Z 992.126,A 0.000,B 0.000,C 90.000,E1 238.614} C_DIS
LIN {X 0.124,Y -503.397,Z 992.121,A 0.000,B 0.000,C 90.000,E1 237.709} C_DIS
LIN {X 0.101,Y -500.244,Z 992.112,A 0.000,B 0.000,C 90.000,E1 236.215} C_DIS
LIN {X 0.014,Y -497.594,Z 992.106,A 0.000,B 0.000,C 90.000,E1 235.022} C_DIS
LIN {X 0.149,Y -494.001,Z 992.097,A 0.000,B 0.000,C 90.000,E1 233.497} C_DIS
LIN {X 0.095,Y -488.858,Z 992.086,A 0.000,B 0.000,C 90.000,E1 231.376} C_DIS
LIN {X 0.122,Y -485.918,Z 992.079,A 0.000,B 0.000,C 90.000,E1 230.150} C_DIS
LIN {X 0.172,Y -482.420,Z 992.070,A 0.000,B 0.000,C 90.000,E1 228.609} C_DIS
LIN {X 0.299,Y -476.361,Z 992.055,A 0.000,B 0.000,C 90.000,E1 225.810} C_DIS
LIN {X 0.157,Y -473.057,Z 992.046,A 0.000,B 0.000,C 90.000,E1 224.271} C_DIS
LIN {X 0.115,Y -471.051,Z 992.041,A 0.000,B 0.000,C 90.000,E1 223.338} C_DIS
LIN {X 0.209,Y -467.528,Z 992.032,A 0.000,B 0.000,C 90.000,E1 221.757} C_DIS
LIN {X -0.142,Y -464.772,Z 992.025,A 0.000,B 0.000,C 90.000,E1 220.539} C_DIS
LIN {X -0.033,Y -460.473,Z 992.015,A 0.000,B 0.000,C 90.000,E1 218.624} C_DIS
LIN {X -0.029,Y -456.261,Z 992.004,A 0.000,B 0.000,C 90.000,E1 216.710} C_DIS
LIN {X 0.066,Y -452.053,Z 991.993,A 0.000,B 0.000,C 90.000,E1 214.771} C_DIS
LIN {X -0.005,Y -448.566,Z 991.984,A 0.000,B 0.000,C 90.000,E1 213.166} C_DIS
LIN {X -0.084,Y -445.721,Z 991.977,A 0.000,B 0.000,C 90.000,E1 211.878} C_DIS
LIN {X -0.153,Y -442.221,Z 991.968,A 0.000,B 0.000,C 90.000,E1 210.256} C_DIS
LIN {X -0.221,Y -440.022,Z 991.963,A 0.000,B 0.000,C 90.000,E1 209.283} C_DIS
LIN {X -0.009,Y -434.884,Z 991.950,A 0.000,B 0.000,C 90.000,E1 206.950} C_DIS
LIN {X 0.050,Y -431.152,Z 991.941,A 0.000,B 0.000,C 90.000,E1 205.283} C_DIS
LIN {X 0.011,Y -425.793,Z 991.928,A 0.000,B 0.000,C 90.000,E1 202.950} C_DIS
LIN {X 0.057,Y -419.934,Z 991.913,A 0.000,B 0.000,C 90.000,E1 200.248} C_DIS
LIN {X -0.206,Y -413.825,Z 991.896,A 0.000,B 0.000,C 90.000,E1 197.221} C_DIS
LIN {X 0.135,Y -408.890,Z 991.880,A 0.000,B 0.000,C 90.000,E1 194.426} C_DIS
LIN {X -0.005,Y -406.557,Z 991.873,A 0.000,B 0.000,C 90.000,E1 193.063} C_DIS
LIN {X 0.204,Y -403.570,Z 991.863,A 0.000,B 0.000,C 90.000,E1 191.299} C_DIS
LIN {X 0.046,Y -397.177,Z 991.842,A 0.000,B 0.000,C 90.000,E1 187.473} C_DIS
LIN {X -0.033,Y -396.343,Z 991.836,A 0.000,B 0.000,C 90.000,E1 186.429} C_DIS
LIN {X -0.139,Y -396.176,Z 991.832,A 0.000,B 0.000,C 90.000,E1 185.739} C_DIS
LIN {X 0.185,Y -396.352,Z 991.829,A 0.000,B 0.000,C 90.000,E1 185.163} C_DIS
LIN {X 0.047,Y -397.834,Z 991.824,A 0.000,B 0.000,C 90.000,E1 184.302} C_DIS
LIN {X 0.011,Y -398.804,Z 991.822,A 0.000,B 0.000,C 90.000,E1 183.955} C_DIS
LIN {X -0.061,Y -400.884,Z 991.819,A 0.000,B 0.000,C 90.000,E1 183.440} C_DIS
LIN {X -0.108,Y -403.128,Z 991.817,A 0.000,B 0.000,C 90.000,E1 183.037} C_DIS
LIN {X -0.169,Y -406.410,Z 991.814,A 0.000,B 0.000,C 90.000,E1 182.522} C_DIS
LIN {X -0.160,Y -411.940,Z 991.810,A 0.000,B 0.000,C 90.000,E1 181.835} C_DIS
LIN {X 0.067,Y -420.539,Z 991.805,A 0.000,B 0.000,C 90.000,E1 180.859} C_DIS
LIN {X -0.063,Y -424.623,Z 991.803,A 0.000,B 0.000,C 90.000,E1 180.458} C_DIS
LIN {X 0.055,Y -437.416,Z 991.795,A 0.000,B 0.000,C 90.000,E1 179.141} C_DIS
LIN {X -0.016,Y -448.712,Z 991.789,A 0.000,B 0.000,C 90.000,E1 177.993} C_DIS
LIN {X -0.038,Y -456.752,Z 991.784,A 0.000,B 0.000,C 90.000,E1 177.135} C_DIS
LIN {X -0.219,Y -462.241,Z 991.781,A 0.000,B 0.000,C 90.000,E1 176.560} C_DIS
LIN {X 0.243,Y -468.697,Z 991.777,A 0.000,B 0.000,C 90.000,E1 175.755} C_DIS
LIN {X 0.071,Y -476.419,Z 991.771,A 0.000,B 0.000,C 90.000,E1 174.837} C_DIS
LIN {X 0.007,Y -483.664,Z 991.766,A 0.000,B 0.000,C 90.000,E1 173.913} C_DIS
LIN {X 0.137,Y -491.230,Z 991.761,A 0.000,B 0.000,C 90.000,E1 172.875} C_DIS
LIN {X 0.005,Y -498.775,Z 991.755,A 0.000,B 0.000,C 90.000,E1 171.837} C_DIS
LIN {X 0.192,Y -504.986,Z 991.750,A 0.000,B 0.000,C 90.000,E1 170.914} C_DIS
LIN {X -0.008,Y -513.027,Z 991.743,A 0.000,B 0.000,C 90.000,E1 169.746} C_DIS
LIN {X 0.135,Y -517.719,Z 991.739,A 0.000,B 0.000,C 90.000,E1 168.993} C_DIS
LIN {X 0.009,Y -524.108,Z 991.733,A 0.000,B 0.000,C 90.000,E1 167.993} C_DIS
LIN {X 0.088,Y -531.153,Z 991.727,A 0.000,B 0.000,C 90.000,E1 166.825} C_DIS
LIN {X 0.228,Y -538.932,Z 991.720,A 0.000,B 0.000,C 90.000,E1 165.519} C_DIS
LIN {X -0.247,Y -544.845,Z 991.714,A 0.000,B 0.000,C 90.000,E1 164.574} C_DIS
LIN {X 0.086,Y -554.513,Z 991.705,A 0.000,B 0.000,C 90.000,E1 162.851} C_DIS
LIN {X -0.177,Y -560.550,Z 991.699,A 0.000,B 0.000,C 90.000,E1 161.764} C_DIS
LIN {X 0.040,Y -565.024,Z 991.694,A 0.000,B 0.000,C 90.000,E1 160.913} C_DIS
LIN {X -0.077,Y -570.747,Z 991.688,A 0.000,B 0.000,C 90.000,E1 159.826} C_DIS
LIN {X 0.165,Y -575.595,Z 991.683,A 0.000,B 0.000,C 90.000,E1 158.847} C_DIS
LIN {X -0.072,Y -580.153,Z 991.677,A 0.000,B 0.000,C 90.000,E1 157.922} C_DIS
LIN {X -0.029,Y -584.375,Z 991.672,A 0.000,B 0.000,C 90.000,E1 156.975} C_DIS
LIN {X -0.044,Y -587.392,Z 991.668,A 0.000,B 0.000,C 90.000,E1 156.305} C_DIS
LIN {X 0.035,Y -591.711,Z 991.662,A 0.000,B 0.000,C 90.000,E1 155.229} C_DIS
LIN {X 0.175,Y -595.642,Z 991.657,A 0.000,B 0.000,C 90.000,E1 154.152} C_DIS
LIN {X -0.086,Y -598.372,Z 991.652,A 0.000,B 0.000,C 90.000,E1 153.384} C_DIS
LIN {X 0.137,Y -601.738,Z 991.646,A 0.000,B 0.000,C 90.000,E1 152.308} C_DIS
LIN {X 0.324,Y -606.377,Z 991.638,A 0.000,B 0.000,C 90.000,E1 150.717} C_DIS
LIN {X -0.113,Y -609.459,Z 991.632,A 0.000,B 0.000,C 90.000,E1 149.715} C_DIS
LIN {X -0.030,Y -613.202,Z 991.625,A 0.000,B 0.000,C 90.000,E1 148.408} C_DIS
LIN {X 0.204,Y -617.589,Z 991.616,A 0.000,B 0.000,C 90.000,E1 146.834} C_DIS
LIN {X -0.195,Y -623.411,Z 991.604,A 0.000,B 0.000,C 90.000,E1 144.815} C_DIS
LIN {X 0.101,Y -627.795,Z 991.596,A 0.000,B 0.000,C 90.000,E1 143.256} C_DIS
LIN {X -0.020,Y -632.087,Z 991.588,A 0.000,B 0.000,C 90.000,E1 141.743} C_DIS
LIN {X -0.041,Y -635.640,Z 991.581,A 0.000,B 0.000,C 90.000,E1 140.481} C_DIS
LIN {X -0.004,Y -639.122,Z 991.573,A 0.000,B 0.000,C 90.000,E1 139.218} C_DIS
LIN {X 0.078,Y -642.536,Z 991.567,A 0.000,B 0.000,C 90.000,E1 137.957} C_DIS
LIN {X -0.038,Y -648.203,Z 991.555,A 0.000,B 0.000,C 90.000,E1 135.972} C_DIS
LIN {X -0.069,Y -655.888,Z 991.542,A 0.000,B 0.000,C 90.000,E1 133.500} C_DIS
LIN {X 0.229,Y -660.878,Z 991.534,A 0.000,B 0.000,C 90.000,E1 132.000} C_DIS
LIN {X 0.177,Y -666.042,Z 991.525,A 0.000,B 0.000,C 90.000,E1 130.539} C_DIS
LIN {X -0.215,Y -670.231,Z 991.519,A 0.000,B 0.000,C 90.000,E1 129.358} C_DIS
LIN {X 0.407,Y -674.083,Z 991.512,A 0.000,B 0.000,C 90.000,E1 128.096} C_DIS
LIN {X -0.274,Y -677.752,Z 991.505,A 0.000,B 0.000,C 90.000,E1 126.950} C_DIS
LIN {X -0.341,Y -681.879,Z 991.497,A 0.000,B 0.000,C 90.000,E1 125.518} C_DIS
LIN {X 0.024,Y -684.599,Z 991.492,A 0.000,B 0.000,C 90.000,E1 124.532} C_DIS
LIN {X 0.040,Y -687.165,Z 991.487,A 0.000,B 0.000,C 90.000,E1 123.579} C_DIS
LIN {X -0.046,Y -691.481,Z 991.477,A 0.000,B 0.000,C 90.000,E1 121.926} C_DIS
LIN {X -0.305,Y -693.913,Z 991.472,A 0.000,B 0.000,C 90.000,E1 121.003} C_DIS
LIN {X -0.177,Y -696.063,Z 991.467,A 0.000,B 0.000,C 90.000,E1 120.050} C_DIS
LIN {X 0.325,Y -697.021,Z 991.464,A 0.000,B 0.000,C 90.000,E1 119.539} C_DIS
LIN {X -0.121,Y -698.242,Z 991.460,A 0.000,B 0.000,C 90.000,E1 118.871} C_DIS
LIN {X 0.053,Y -699.175,Z 991.456,A 0.000,B 0.000,C 90.000,E1 118.153} C_DIS
LIN {X -0.359,Y -699.708,Z 991.454,A 0.000,B 0.000,C 90.000,E1 117.719} C_DIS
LIN {X -0.016,Y -701.104,Z 991.445,A 0.000,B 0.000,C 90.000,E1 116.052} C_DIS
LIN {X 0.178,Y -701.676,Z 991.441,A 0.000,B 0.000,C 90.000,E1 115.335} C_DIS
LIN {X -0.305,Y -701.960,Z 991.434,A 0.000,B 0.000,C 90.000,E1 114.207} C_DIS
LIN {X 0.243,Y -701.505,Z 991.432,A 0.000,B 0.000,C 90.000,E1 113.695} C_DIS
LIN {X 0.236,Y -701.074,Z 991.430,A 0.000,B 0.000,C 90.000,E1 113.462} C_DIS
LIN {X -0.008,Y -698.467,Z 991.427,A 0.000,B 0.000,C 90.000,E1 112.898} C_DIS
LIN {X 0.124,Y -697.632,Z 991.427,A 0.000,B 0.000,C 90.000,E1 112.770} C_DIS
LIN {X -0.337,Y -693.899,Z 991.425,A 0.000,B 0.000,C 90.000,E1 112.461} C_DIS
LIN {X 0.084,Y -691.153,Z 991.423,A 0.000,B 0.000,C 90.000,E1 112.206} C_DIS
LIN {X 0.312,Y -688.803,Z 991.423,A 0.000,B 0.000,C 90.000,E1 112.078} C_DIS
LIN {X -0.201,Y -684.560,Z 991.422,A 0.000,B 0.000,C 90.000,E1 111.972} C_DIS
LIN {X -0.285,Y -677.207,Z 991.421,A 0.000,B 0.000,C 90.000,E1 111.844} C_DIS
LIN {X 0.189,Y -674.845,Z 991.421,A 0.000,B 0.000,C 90.000,E1 111.770} C_DIS
LIN {X 0.143,Y -670.173,Z 991.421,A 0.000,B 0.000,C 90.000,E1 111.770} C_DIS
LIN {X 0.089,Y -620.719,Z 991.421,A 0.000,B 0.000,C 90.000,E1 111.770} C_DIS
LIN {X -0.176,Y -616.949,Z 991.421,A 0.000,B 0.000,C 90.000,E1 111.716} C_DIS
LIN {X 0.159,Y -609.946,Z 991.419,A 0.000,B 0.000,C 90.000,E1 111.482} C_DIS
LIN {X 0.148,Y -602.344,Z 991.418,A 0.000,B 0.000,C 90.000,E1 111.173} C_DIS
LIN {X -0.056,Y -595.234,Z 991.416,A 0.000,B 0.000,C 90.000,E1 110.791} C_DIS
LIN {X 0.110,Y -590.934,Z 991.414,A 0.000,B 0.000,C 90.000,E1 110.482} C_DIS
LIN {X 0.142,Y -581.668,Z 991.410,A 0.000,B 0.000,C 90.000,E1 109.758} C_DIS
LIN {X -0.071,Y -575.846,Z 991.407,A 0.000,B 0.000,C 90.000,E1 109.322} C_DIS
LIN {X 0.118,Y -573.019,Z 991.406,A 0.000,B 0.000,C 90.000,E1 109.087} C_DIS
LIN {X -0.186,Y -566.620,Z 991.404,A 0.000,B 0.000,C 90.000,E1 108.725} C_DIS
LIN {X -0.247,Y -563.068,Z 991.403,A 0.000,B 0.000,C 90.000,E1 108.544} C_DIS
LIN {X -0.029,Y -551.358,Z 991.400,A 0.000,B 0.000,C 90.000,E1 107.946} C_DIS
LIN {X -0.021,Y -550.508,Z 991.399,A 0.000,B 0.000,C 90.000,E1 107.873} C_DIS
LIN {X -0.273,Y -549.247,Z 991.399,A 0.000,B 0.000,C 90.000,E1 107.764} C_DIS
LIN {X -0.314,Y -549.231,Z 991.399,A 0.000,B 0.000,C 90.000,E1 107.764} C_DIS
LIN {X 0.149,Y -548.818,Z 991.397,A 0.000,B 0.000,C 90.000,E1 107.511} C_DIS
LIN {X -0.193,Y -548.771,Z 991.394,A 0.000,B 0.000,C 90.000,E1 106.985} C_DIS
LIN {X -0.025,Y -549.286,Z 991.388,A 0.000,B 0.000,C 90.000,E1 105.843} C_DIS
LIN {X -0.082,Y -550.246,Z 991.377,A 0.000,B 0.000,C 90.000,E1 103.883} C_DIS
LIN {X -0.204,Y -553.152,Z 991.357,A 0.000,B 0.000,C 90.000,E1 100.254} C_DIS
LIN {X -0.106,Y -554.935,Z 991.348,A 0.000,B 0.000,C 90.000,E1 98.568} C_DIS
LIN {X -0.056,Y -556.711,Z 991.338,A 0.000,B 0.000,C 90.000,E1 96.891} C_DIS
LIN {X -0.232,Y -557.751,Z 991.332,A 0.000,B 0.000,C 90.000,E1 95.796} C_DIS
LIN {X 0.240,Y -558.733,Z 991.324,A 0.000,B 0.000,C 90.000,E1 94.359} C_DIS
LIN {X 0.053,Y -559.381,Z 991.318,A 0.000,B 0.000,C 90.000,E1 93.269} C_DIS
LIN {X -0.033,Y -560.128,Z 991.311,A 0.000,B 0.000,C 90.000,E1 91.892} C_DIS
LIN {X -0.015,Y -560.995,Z 991.301,A 0.000,B 0.000,C 90.000,E1 90.229} C_DIS
LIN {X -0.091,Y -561.599,Z 991.294,A 0.000,B 0.000,C 90.000,E1 88.854} C_DIS
LIN {X -0.147,Y -561.902,Z 991.286,A 0.000,B 0.000,C 90.000,E1 87.478} C_DIS
LIN {X 0.028,Y -562.222,Z 991.275,A 0.000,B 0.000,C 90.000,E1 85.527} C_DIS
LIN {X 0.248,Y -562.478,Z 991.264,A 0.000,B 0.000,C 90.000,E1 83.571} C_DIS
LIN {X 0.052,Y -562.864,Z 991.254,A 0.000,B 0.000,C 90.000,E1 81.659} C_DIS
LIN {X -0.129,Y -563.443,Z 991.243,A 0.000,B 0.000,C 90.000,E1 79.746} C_DIS
LIN {X 0.132,Y -564.075,Z 991.235,A 0.000,B 0.000,C 90.000,E1 78.342} C_DIS
LIN {X 0.020,Y -564.928,Z 991.226,A 0.000,B 0.000,C 90.000,E1 76.700} C_DIS
LIN {X 0.153,Y -566.566,Z 991.212,A 0.000,B 0.000,C 90.000,E1 74.212} C_DIS
LIN {X -0.174,Y -567.770,Z 991.203,A 0.000,B 0.000,C 90.000,E1 72.598} C_DIS
LIN {X -0.107,Y -568.748,Z 991.196,A 0.000,B 0.000,C 90.000,E1 71.221} C_DIS
LIN {X 0.151,Y -569.580,Z 991.188,A 0.000,B 0.000,C 90.000,E1 69.826} C_DIS
LIN {X 0.093,Y -570.355,Z 991.180,A 0.000,B 0.000,C 90.000,E1 68.465} C_DIS
LIN {X -0.116,Y -571.165,Z 991.171,A 0.000,B 0.000,C 90.000,E1 66.847} C_DIS
LIN {X 0.023,Y -571.573,Z 991.165,A 0.000,B 0.000,C 90.000,E1 65.741} C_DIS
LIN {X -0.128,Y -572.020,Z 991.159,A 0.000,B 0.000,C 90.000,E1 64.665} C_DIS
LIN {X 0.169,Y -572.493,Z 991.150,A 0.000,B 0.000,C 90.000,E1 62.999} C_DIS
LIN {X 0.128,Y -572.827,Z 991.143,A 0.000,B 0.000,C 90.000,E1 61.641} C_DIS
LIN {X 0.085,Y -573.141,Z 991.135,A 0.000,B 0.000,C 90.000,E1 60.284} C_DIS
LIN {X -0.171,Y -573.364,Z 991.127,A 0.000,B 0.000,C 90.000,E1 58.948} C_DIS
LIN {X 0.020,Y -573.567,Z 991.118,A 0.000,B 0.000,C 90.000,E1 57.296} C_DIS
LIN {X 0.089,Y -573.694,Z 991.111,A 0.000,B 0.000,C 90.000,E1 55.928} C_DIS
LIN {X 0.004,Y -573.733,Z 991.105,A 0.000,B 0.000,C 90.000,E1 54.848} C_DIS
LIN {X -0.082,Y -573.503,Z 991.097,A 0.000,B 0.000,C 90.000,E1 53.497} C_DIS
LIN {X 0.035,Y -573.079,Z 991.091,A 0.000,B 0.000,C 90.000,E1 52.396} C_DIS
LIN {X -0.345,Y -572.693,Z 991.087,A 0.000,B 0.000,C 90.000,E1 51.618} C_DIS
LIN {X -0.239,Y -571.981,Z 991.081,A 0.000,B 0.000,C 90.000,E1 50.517} C_DIS
LIN {X 0.091,Y -571.342,Z 991.076,A 0.000,B 0.000,C 90.000,E1 49.666} C_DIS
LIN {X 0.171,Y -570.269,Z 991.070,A 0.000,B 0.000,C 90.000,E1 48.566} C_DIS
LIN {X 0.063,Y -569.324,Z 991.065,A 0.000,B 0.000,C 90.000,E1 47.757} C_DIS
LIN {X -0.015,Y -568.205,Z 991.061,A 0.000,B 0.000,C 90.000,E1 46.944} C_DIS
LIN {X -0.136,Y -566.867,Z 991.056,A 0.000,B 0.000,C 90.000,E1 46.134} C_DIS
LIN {X -0.266,Y -565.378,Z 991.052,A 0.000,B 0.000,C 90.000,E1 45.324} C_DIS
LIN {X -0.015,Y -563.667,Z 991.047,A 0.000,B 0.000,C 90.000,E1 44.474} C_DIS
LIN {X 0.222,Y -561.728,Z 991.043,A 0.000,B 0.000,C 90.000,E1 43.623} C_DIS
LIN {X -0.020,Y -560.310,Z 991.039,A 0.000,B 0.000,C 90.000,E1 43.095} C_DIS
LIN {X -0.146,Y -557.109,Z 991.033,A 0.000,B 0.000,C 90.000,E1 42.000} C_DIS
LIN {X 0.025,Y -554.305,Z 991.029,A 0.000,B 0.000,C 90.000,E1 41.148} C_DIS
LIN {X -0.259,Y -552.323,Z 991.026,A 0.000,B 0.000,C 90.000,E1 40.620} C_DIS
LIN {X 0.277,Y -548.921,Z 991.021,A 0.000,B 0.000,C 90.000,E1 39.725} C_DIS
LIN {X 0.002,Y -545.185,Z 991.016,A 0.000,B 0.000,C 90.000,E1 38.910} C_DIS
LIN {X -0.317,Y -541.135,Z 991.012,A 0.000,B 0.000,C 90.000,E1 38.096} C_DIS
LIN {X -0.097,Y -537.590,Z 991.008,A 0.000,B 0.000,C 90.000,E1 37.363} C_DIS
LIN {X -0.078,Y -531.523,Z 991.001,A 0.000,B 0.000,C 90.000,E1 36.217} C_DIS
LIN {X -0.265,Y -527.499,Z 990.997,A 0.000,B 0.000,C 90.000,E1 35.518} C_DIS
LIN {X 0.112,Y -524.092,Z 990.994,A 0.000,B 0.000,C 90.000,E1 34.898} C_DIS
LIN {X -0.192,Y -517.678,Z 990.988,A 0.000,B 0.000,C 90.000,E1 33.913} C_DIS
LIN {X 0.107,Y -513.844,Z 990.985,A 0.000,B 0.000,C 90.000,E1 33.293} C_DIS
LIN {X 0.098,Y -509.742,Z 990.982,A 0.000,B 0.000,C 90.000,E1 32.704} C_DIS
LIN {X -0.094,Y -505.279,Z 990.979,A 0.000,B 0.000,C 90.000,E1 32.133} C_DIS
LIN {X -0.089,Y -499.358,Z 990.974,A 0.000,B 0.000,C 90.000,E1 31.386} C_DIS
LIN {X -0.193,Y -494.251,Z 990.971,A 0.000,B 0.000,C 90.000,E1 30.797} C_DIS
LIN {X -0.178,Y -488.909,Z 990.968,A 0.000,B 0.000,C 90.000,E1 30.207} C_DIS
LIN {X -0.096,Y -479.056,Z 990.962,A 0.000,B 0.000,C 90.000,E1 29.205} C_DIS
LIN {X 0.042,Y -471.835,Z 990.958,A 0.000,B 0.000,C 90.000,E1 28.487} C_DIS
LIN {X 0.246,Y -461.532,Z 990.953,A 0.000,B 0.000,C 90.000,E1 27.513} C_DIS
LIN {X 0.035,Y -450.999,Z 990.948,A 0.000,B 0.000,C 90.000,E1 26.616} C_DIS
LIN {X 0.118,Y -438.970,Z 990.942,A 0.000,B 0.000,C 90.000,E1 25.591} C_DIS
LIN {X 0.134,Y -418.214,Z 990.932,A 0.000,B 0.000,C 90.000,E1 23.695} C_DIS
LIN {X 0.247,Y -403.737,Z 990.924,A 0.000,B 0.000,C 90.000,E1 22.206} C_DIS
LIN {X -0.007,Y -399.504,Z 990.921,A 0.000,B 0.000,C 90.000,E1 21.770} C_DIS
LIN {X 0.075,Y -395.041,Z 990.918,A 0.000,B 0.000,C 90.000,E1 21.173} C_DIS
LIN {X -0.114,Y -393.855,Z 990.917,A 0.000,B 0.000,C 90.000,E1 21.025} C_DIS
LIN {X 0.065,Y -392.059,Z 990.915,A 0.000,B 0.000,C 90.000,E1 20.663} C_DIS
LIN {X 0.156,Y -391.581,Z 990.914,A 0.000,B 0.000,C 90.000,E1 20.429} C_DIS
LIN {X -0.163,Y -390.598,Z 990.912,A 0.000,B 0.000,C 90.000,E1 20.120} C_DIS
LIN {X -0.072,Y -390.072,Z 990.908,A 0.000,B 0.000,C 90.000,E1 19.396} C_DIS
LIN {X -0.117,Y -390.507,Z 990.903,A 0.000,B 0.000,C 90.000,E1 18.489} C_DIS
LIN {X 0.196,Y -393.747,Z 990.885,A 0.000,B 0.000,C 90.000,E1 15.245} C_DIS
LIN {X 0.163,Y -398.724,Z 990.863,A 0.000,B 0.000,C 90.000,E1 11.366} C_DIS
LIN {X 0.129,Y -404.490,Z 990.844,A 0.000,B 0.000,C 90.000,E1 7.871} C_DIS
LIN {X 0.041,Y -409.191,Z 990.830,A 0.000,B 0.000,C 90.000,E1 5.454} C_DIS
LIN {X 0.088,Y -414.373,Z 990.817,A 0.000,B 0.000,C 90.000,E1 3.037} C_DIS
LIN {X 0.144,Y -417.333,Z 990.809,A 0.000,B 0.000,C 90.000,E1 1.661} C_DIS
LIN {X 0.184,Y -419.223,Z 990.806,A 0.000,B 0.000,C 90.000,E1 0.974} C_DIS
LIN {X 0.197,Y -419.866,Z 990.805,A 0.000,B 0.000,C 90.000,E1 0.802} C_DIS
LIN {X -0.089,Y -423.006,Z 990.801,A 0.000,B 0.000,C 90.000,E1 0.172} C_DIS
LIN {X 0.000,Y -424.198,Z 990.800,A 0.000,B 0.000,C 90.000,E1 360.000} C_DIS
LIN {X -0.100,Y -427.551,Z 990.798,A 0.000,B 0.000,C 90.000,E1 359.656} C_DIS
LIN {X 0.066,Y -428.924,Z 990.797,A 0.000,B 0.000,C 90.000,E1 359.484} C_DIS
LIN {X -0.032,Y -434.106,Z 990.795,A 0.000,B 0.000,C 90.000,E1 359.141} C_DIS
LIN {X 0.063,Y -450.399,Z 990.790,A 0.000,B 0.000,C 90.000,E1 358.224} C_DIS
LIN {X 0.087,Y -463.636,Z 990.786,A 0.000,B 0.000,C 90.000,E1 357.478} C_DIS
LIN {X 0.170,Y -478.588,Z 990.781,A 0.000,B 0.000,C 90.000,E1 356.617} C_DIS
LIN {X 0.137,Y -486.889,Z 990.779,A 0.000,B 0.000,C 90.000,E1 356.159} C_DIS
LIN {X -0.190,Y -498.355,Z 990.775,A 0.000,B 0.000,C 90.000,E1 355.527} C_DIS
LIN {X -0.187,Y -509.476,Z 990.771,A 0.000,B 0.000,C 90.000,E1 354.837} C_DIS
LIN {X -0.090,Y -518.727,Z 990.768,A 0.000,B 0.000,C 90.000,E1 354.204} C_DIS
LIN {X 0.143,Y -526.321,Z 990.765,A 0.000,B 0.000,C 90.000,E1 353.628} C_DIS
LIN {X 0.162,Y -533.647,Z 990.762,A 0.000,B 0.000,C 90.000,E1 353.053} C_DIS
LIN {X -0.022,Y -539.337,Z 990.759,A 0.000,B 0.000,C 90.000,E1 352.591} C_DIS
LIN {X -0.024,Y -547.210,Z 990.755,A 0.000,B 0.000,C 90.000,E1 351.837} C_DIS
LIN {X -0.097,Y -552.436,Z 990.752,A 0.000,B 0.000,C 90.000,E1 351.310} C_DIS
LIN {X 0.137,Y -557.350,Z 990.749,A 0.000,B 0.000,C 90.000,E1 350.735} C_DIS
LIN {X 0.165,Y -562.919,Z 990.745,A 0.000,B 0.000,C 90.000,E1 350.038} C_DIS
LIN {X 0.241,Y -567.948,Z 990.741,A 0.000,B 0.000,C 90.000,E1 349.342} C_DIS
LIN {X 0.040,Y -571.591,Z 990.738,A 0.000,B 0.000,C 90.000,E1 348.814} C_DIS
LIN {X 0.125,Y -576.515,Z 990.733,A 0.000,B 0.000,C 90.000,E1 347.993} C_DIS
LIN {X -0.250,Y -580.302,Z 990.730,A 0.000,B 0.000,C 90.000,E1 347.353} C_DIS
LIN {X -0.235,Y -585.280,Z 990.724,A 0.000,B 0.000,C 90.000,E1 346.408} C_DIS
LIN {X 0.333,Y -590.646,Z 990.718,A 0.000,B 0.000,C 90.000,E1 345.283} C_DIS
LIN {X -0.092,Y -595.101,Z 990.713,A 0.000,B 0.000,C 90.000,E1 344.393} C_DIS
LIN {X -0.016,Y -600.501,Z 990.707,A 0.000,B 0.000,C 90.000,E1 343.196} C_DIS
LIN {X 0.180,Y -604.933,Z 990.701,A 0.000,B 0.000,C 90.000,E1 342.127} C_DIS
LIN {X 0.044,Y -609.216,Z 990.695,A 0.000,B 0.000,C 90.000,E1 341.094} C_DIS
LIN {X -0.032,Y -613.172,Z 990.689,A 0.000,B 0.000,C 90.000,E1 340.061} C_DIS
LIN {X 0.198,Y -615.876,Z 990.685,A 0.000,B 0.000,C 90.000,E1 339.263} C_DIS
LIN {X 0.185,Y -620.122,Z 990.678,A 0.000,B 0.000,C 90.000,E1 337.975} C_DIS
LIN {X -0.343,Y -624.041,Z 990.671,A 0.000,B 0.000,C 90.000,E1 336.741} C_DIS
LIN {X 0.265,Y -627.598,Z 990.664,A 0.000,B 0.000,C 90.000,E1 335.409} C_DIS
LIN {X 0.082,Y -630.280,Z 990.658,A 0.000,B 0.000,C 90.000,E1 334.409} C_DIS
LIN {X 0.169,Y -632.122,Z 990.654,A 0.000,B 0.000,C 90.000,E1 333.640} C_DIS
LIN {X 0.314,Y -634.329,Z 990.648,A 0.000,B 0.000,C 90.000,E1 332.615} C_DIS
LIN {X 0.017,Y -637.391,Z 990.640,A 0.000,B 0.000,C 90.000,E1 331.129} C_DIS
LIN {X 0.080,Y -640.132,Z 990.631,A 0.000,B 0.000,C 90.000,E1 329.616} C_DIS
LIN {X 0.076,Y -641.822,Z 990.626,A 0.000,B 0.000,C 90.000,E1 328.614} C_DIS
LIN {X 0.091,Y -643.245,Z 990.620,A 0.000,B 0.000,C 90.000,E1 327.612} C_DIS
LIN {X -0.069,Y -644.559,Z 990.615,A 0.000,B 0.000,C 90.000,E1 326.628} C_DIS
LIN {X 0.335,Y -645.623,Z 990.609,A 0.000,B 0.000,C 90.000,E1 325.595} C_DIS
LIN {X -0.256,Y -646.676,Z 990.602,A 0.000,B 0.000,C 90.000,E1 324.402} C_DIS
LIN {X 0.072,Y -647.557,Z 990.595,A 0.000,B 0.000,C 90.000,E1 323.130} C_DIS
LIN {X -0.028,Y -648.045,Z 990.590,A 0.000,B 0.000,C 90.000,E1 322.145} C_DIS
LIN {X -0.358,Y -648.783,Z 990.580,A 0.000,B 0.000,C 90.000,E1 320.436} C_DIS
LIN {X -0.119,Y -649.261,Z 990.573,A 0.000,B 0.000,C 90.000,E1 319.175} C_DIS
LIN {X -0.223,Y -650.965,Z 990.558,A 0.000,B 0.000,C 90.000,E1 316.458} C_DIS
LIN {X -0.058,Y -651.933,Z 990.550,A 0.000,B 0.000,C 90.000,E1 314.960} C_DIS
LIN {X 0.036,Y -653.454,Z 990.539,A 0.000,B 0.000,C 90.000,E1 312.975} C_DIS
LIN {X -0.145,Y -654.346,Z 990.532,A 0.000,B 0.000,C 90.000,E1 311.757} C_DIS
LIN {X 0.147,Y -655.280,Z 990.524,A 0.000,B 0.000,C 90.000,E1 310.253} C_DIS
LIN {X 0.044,Y -656.030,Z 990.516,A 0.000,B 0.000,C 90.000,E1 308.785} C_DIS
LIN {X -0.042,Y -656.652,Z 990.507,A 0.000,B 0.000,C 90.000,E1 307.317} C_DIS
LIN {X 0.380,Y -656.965,Z 990.502,A 0.000,B 0.000,C 90.000,E1 306.297} C_DIS
LIN {X -0.111,Y -657.166,Z 990.494,A 0.000,B 0.000,C 90.000,E1 304.865} C_DIS
LIN {X 0.110,Y -657.490,Z 990.486,A 0.000,B 0.000,C 90.000,E1 303.372} C_DIS
LIN {X -0.196,Y -663.988,Z 990.447,A 0.000,B 0.000,C 90.000,E1 296.539} C_DIS
LIN {X 0.243,Y -665.948,Z 990.441,A 0.000,B 0.000,C 90.000,E1 295.283} C_DIS
LIN {X 0.117,Y -667.787,Z 990.434,A 0.000,B 0.000,C 90.000,E1 294.079} C_DIS
LIN {X -0.146,Y -669.097,Z 990.428,A 0.000,B 0.000,C 90.000,E1 293.131} C_DIS
LIN {X 0.059,Y -669.707,Z 990.424,A 0.000,B 0.000,C 90.000,E1 292.386} C_DIS
LIN {X 0.116,Y -669.755,Z 990.422,A 0.000,B 0.000,C 90.000,E1 291.897} C_DIS
LIN {X 0.176,Y -669.245,Z 990.419,A 0.000,B 0.000,C 90.000,E1 291.408} C_DIS
LIN {X 0.085,Y -668.845,Z 990.418,A 0.000,B 0.000,C 90.000,E1 291.173} C_DIS
LIN {X 0.308,Y -667.162,Z 990.416,A 0.000,B 0.000,C 90.000,E1 290.791} C_DIS
LIN {X 0.214,Y -665.829,Z 990.414,A 0.000,B 0.000,C 90.000,E1 290.556} C_DIS
LIN {X 0.284,Y -664.969,Z 990.414,A 0.000,B 0.000,C 90.000,E1 290.429} C_DIS
LIN {X 0.350,Y -663.863,Z 990.413,A 0.000,B 0.000,C 90.000,E1 290.301} C_DIS
LIN {X 0.119,Y -657.980,Z 990.411,A 0.000,B 0.000,C 90.000,E1 289.885} C_DIS
LIN {X 0.226,Y -650.241,Z 990.408,A 0.000,B 0.000,C 90.000,E1 289.396} C_DIS
LIN {X -0.341,Y -646.364,Z 990.407,A 0.000,B 0.000,C 90.000,E1 289.214} C_DIS
LIN {X 0.241,Y -644.240,Z 990.406,A 0.000,B 0.000,C 90.000,E1 288.960} C_DIS
LIN {X 0.196,Y -644.206,Z 990.405,A 0.000,B 0.000,C 90.000,E1 288.960} C_DIS
LIN {X 0.221,Y -644.295,Z 990.404,A 0.000,B 0.000,C 90.000,E1 288.779} C_DIS
LIN {X -0.061,Y -646.306,Z 990.402,A 0.000,B 0.000,C 90.000,E1 288.362} C_DIS
LIN {X 0.250,Y -653.925,Z 990.395,A 0.000,B 0.000,C 90.000,E1 287.094} C_DIS
LIN {X -0.108,Y -657.977,Z 990.391,A 0.000,B 0.000,C 90.000,E1 286.386} C_DIS
LIN {X -0.284,Y -660.746,Z 990.388,A 0.000,B 0.000,C 90.000,E1 285.788} C_DIS
LIN {X 0.331,Y -662.539,Z 990.385,A 0.000,B 0.000,C 90.000,E1 285.245} C_DIS
LIN {X 0.144,Y -663.941,Z 990.382,A 0.000,B 0.000,C 90.000,E1 284.773} C_DIS
LIN {X -0.033,Y -665.045,Z 990.379,A 0.000,B 0.000,C 90.000,E1 284.300} C_DIS
LIN {X -0.201,Y -665.885,Z 990.377,A 0.000,B 0.000,C 90.000,E1 283.828} C_DIS
LIN {X 0.202,Y -666.758,Z 990.373,A 0.000,B 0.000,C 90.000,E1 283.063} C_DIS
LIN {X 0.044,Y -667.107,Z 990.370,A 0.000,B 0.000,C 90.000,E1 282.591} C_DIS
LIN {X -0.114,Y -667.278,Z 990.367,A 0.000,B 0.000,C 90.000,E1 282.119} C_DIS
LIN {X 0.167,Y -667.107,Z 990.363,A 0.000,B 0.000,C 90.000,E1 281.366} C_DIS
LIN {X 0.006,Y -666.828,Z 990.361,A 0.000,B 0.000,C 90.000,E1 280.894} C_DIS
LIN {X -0.161,Y -666.327,Z 990.358,A 0.000,B 0.000,C 90.000,E1 280.423} C_DIS
LIN {X 0.206,Y -665.542,Z 990.355,A 0.000,B 0.000,C 90.000,E1 279.905} C_DIS
LIN {X -0.176,Y -663.858,Z 990.351,A 0.000,B 0.000,C 90.000,E1 279.208} C_DIS
LIN {X 0.184,Y -662.431,Z 990.348,A 0.000,B 0.000,C 90.000,E1 278.690} C_DIS
LIN {X -0.023,Y -660.648,Z 990.346,A 0.000,B 0.000,C 90.000,E1 278.219} C_DIS
LIN {X 0.213,Y -657.946,Z 990.342,A 0.000,B 0.000,C 90.000,E1 277.587} C_DIS
LIN {X -0.117,Y -655.281,Z 990.340,A 0.000,B 0.000,C 90.000,E1 277.125} C_DIS
LIN {X 0.152,Y -651.282,Z 990.336,A 0.000,B 0.000,C 90.000,E1 276.486} C_DIS
LIN {X -0.223,Y -647.527,Z 990.333,A 0.000,B 0.000,C 90.000,E1 276.024} C_DIS
LIN {X -0.099,Y -642.198,Z 990.330,A 0.000,B 0.000,C 90.000,E1 275.391} C_DIS
LIN {X 0.176,Y -638.737,Z 990.328,A 0.000,B 0.000,C 90.000,E1 274.992} C_DIS
LIN {X 0.067,Y -632.783,Z 990.325,A 0.000,B 0.000,C 90.000,E1 274.416} C_DIS
LIN {X -0.033,Y -626.069,Z 990.321,A 0.000,B 0.000,C 90.000,E1 273.841} C_DIS
LIN {X 0.112,Y -618.846,Z 990.318,A 0.000,B 0.000,C 90.000,E1 273.269} C_DIS
LIN {X 0.244,Y -611.406,Z 990.315,A 0.000,B 0.000,C 90.000,E1 272.751} C_DIS
LIN {X -0.263,Y -605.014,Z 990.313,A 0.000,B 0.000,C 90.000,E1 272.407} C_DIS
LIN {X 0.153,Y -598.192,Z 990.311,A 0.000,B 0.000,C 90.000,E1 272.007} C_DIS
LIN {X -0.059,Y -591.260,Z 990.310,A 0.000,B 0.000,C 90.000,E1 271.718} C_DIS
LIN {X 0.082,Y -585.530,Z 990.308,A 0.000,B 0.000,C 90.000,E1 271.489} C_DIS
LIN {X -0.002,Y -578.029,Z 990.307,A 0.000,B 0.000,C 90.000,E1 271.260} C_DIS
LIN {X -0.211,Y -570.235,Z 990.306,A 0.000,B 0.000,C 90.000,E1 271.088} C_DIS
LIN {X -0.224,Y -563.994,Z 990.305,A 0.000,B 0.000,C 90.000,E1 270.974} C_DIS
LIN {X -0.178,Y -557.969,Z 990.305,A 0.000,B 0.000,C 90.000,E1 270.917} C_DIS
LIN {X -0.216,Y -542.957,Z 990.305,A 0.000,B 0.000,C 90.000,E1 270.917} C_DIS
LIN {X -0.089,Y -542.288,Z 990.301,A 0.000,B 0.000,C 90.000,E1 270.229} C_DIS
LIN {X 0.045,Y -541.310,Z 990.293,A 0.000,B 0.000,C 90.000,E1 268.797} C_DIS
LIN {X 0.189,Y -540.164,Z 990.284,A 0.000,B 0.000,C 90.000,E1 267.078} C_DIS
LIN {X -0.203,Y -538.930,Z 990.274,A 0.000,B 0.000,C 90.000,E1 265.412} C_DIS
LIN {X -0.090,Y -537.983,Z 990.268,A 0.000,B 0.000,C 90.000,E1 264.261} C_DIS
LIN {X 0.009,Y -537.009,Z 990.262,A 0.000,B 0.000,C 90.000,E1 263.109} C_DIS
LIN {X 0.159,Y -535.948,Z 990.255,A 0.000,B 0.000,C 90.000,E1 261.951} C_DIS
LIN {X -0.164,Y -533.891,Z 990.244,A 0.000,B 0.000,C 90.000,E1 259.982} C_DIS
LIN {X 0.125,Y -532.064,Z 990.235,A 0.000,B 0.000,C 90.000,E1 258.229} C_DIS
LIN {X -0.226,Y -530.808,Z 990.228,A 0.000,B 0.000,C 90.000,E1 257.117} C_DIS
LIN {X 0.100,Y -528.766,Z 990.219,A 0.000,B 0.000,C 90.000,E1 255.353} C_DIS
LIN {X -0.168,Y -525.955,Z 990.204,A 0.000,B 0.000,C 90.000,E1 252.779} C_DIS
LIN {X 0.166,Y -524.612,Z 990.198,A 0.000,B 0.000,C 90.000,E1 251.583} C_DIS
LIN {X 0.128,Y -522.775,Z 990.190,A 0.000,B 0.000,C 90.000,E1 250.134} C_DIS
LIN {X -0.254,Y -520.922,Z 990.182,A 0.000,B 0.000,C 90.000,E1 248.720} C_DIS
LIN {X 0.012,Y -519.035,Z 990.174,A 0.000,B 0.000,C 90.000,E1 247.230} C_DIS
LIN {X 0.104,Y -517.413,Z 990.167,A 0.000,B 0.000,C 90.000,E1 246.049} C_DIS
LIN {X -0.086,Y -515.701,Z 990.161,A 0.000,B 0.000,C 90.000,E1 244.897} C_DIS
LIN {X -0.055,Y -513.814,Z 990.154,A 0.000,B 0.000,C 90.000,E1 243.717} C_DIS
LIN {X 0.044,Y -511.508,Z 990.146,A 0.000,B 0.000,C 90.000,E1 242.231} C_DIS
LIN {X 0.096,Y -509.078,Z 990.138,A 0.000,B 0.000,C 90.000,E1 240.745} C_DIS
LIN {X -0.051,Y -507.560,Z 990.133,A 0.000,B 0.000,C 90.000,E1 239.871} C_DIS
LIN {X -0.264,Y -504.812,Z 990.124,A 0.000,B 0.000,C 90.000,E1 238.408} C_DIS
LIN {X -0.264,Y -501.720,Z 990.116,A 0.000,B 0.000,C 90.000,E1 236.914} C_DIS
LIN {X -0.046,Y -498.479,Z 990.108,A 0.000,B 0.000,C 90.000,E1 235.388} C_DIS
LIN {X -0.027,Y -496.358,Z 990.103,A 0.000,B 0.000,C 90.000,E1 234.482} C_DIS
LIN {X -0.024,Y -492.769,Z 990.094,A 0.000,B 0.000,C 90.000,E1 232.970} C_DIS
LIN {X -0.244,Y -488.397,Z 990.084,A 0.000,B 0.000,C 90.000,E1 231.170} C_DIS
LIN {X -0.001,Y -482.669,Z 990.071,A 0.000,B 0.000,C 90.000,E1 228.690} C_DIS
LIN {X 0.136,Y -476.588,Z 990.055,A 0.000,B 0.000,C 90.000,E1 225.891} C_DIS
LIN {X 0.192,Y -471.996,Z 990.043,A 0.000,B 0.000,C 90.000,E1 223.704} C_DIS
LIN {X -0.017,Y -468.459,Z 990.034,A 0.000,B 0.000,C 90.000,E1 222.162} C_DIS
LIN {X -0.043,Y -465.678,Z 990.027,A 0.000,B 0.000,C 90.000,E1 220.906} C_DIS
LIN {X 0.118,Y -460.662,Z 990.015,A 0.000,B 0.000,C 90.000,E1 218.669} C_DIS
LIN {X 0.109,Y -457.188,Z 990.006,A 0.000,B 0.000,C 90.000,E1 217.076} C_DIS
LIN {X -0.079,Y -451.547,Z 989.992,A 0.000,B 0.000,C 90.000,E1 214.532} C_DIS
LIN {X -0.094,Y -447.377,Z 989.981,A 0.000,B 0.000,C 90.000,E1 212.594} C_DIS
LIN {X -0.248,Y -442.432,Z 989.968,A 0.000,B 0.000,C 90.000,E1 210.335} C_DIS
LIN {X -0.222,Y -438.735,Z 989.959,A 0.000,B 0.000,C 90.000,E1 208.693} C_DIS
LIN {X -0.065,Y -434.375,Z 989.948,A 0.000,B 0.000,C 90.000,E1 206.693} C_DIS
LIN {X 0.171,Y -431.398,Z 989.941,A 0.000,B 0.000,C 90.000,E1 205.335} C_DIS
LIN {X -0.073,Y -425.221,Z 989.926,A 0.000,B 0.000,C 90.000,E1 202.695} C_DIS
LIN {X -0.050,Y -419.425,Z 989.911,A 0.000,B 0.000,C 90.000,E1 199.993} C_DIS
LIN {X -0.093,Y -413.993,Z 989.896,A 0.000,B 0.000,C 90.000,E1 197.275} C_DIS
LIN {X -0.032,Y -408.457,Z 989.879,A 0.000,B 0.000,C 90.000,E1 194.175} C_DIS
LIN {X 0.215,Y -405.478,Z 989.869,A 0.000,B 0.000,C 90.000,E1 192.411} C_DIS
LIN {X -0.159,Y -402.994,Z 989.861,A 0.000,B 0.000,C 90.000,E1 191.074} C_DIS
LIN {X 0.149,Y -397.019,Z 989.842,A 0.000,B 0.000,C 90.000,E1 187.530} C_DIS
LIN {X 0.098,Y -396.248,Z 989.838,A 0.000,B 0.000,C 90.000,E1 186.834} C_DIS
LIN {X -0.042,Y -395.654,Z 989.832,A 0.000,B 0.000,C 90.000,E1 185.796} C_DIS
LIN {X -0.095,Y -395.751,Z 989.828,A 0.000,B 0.000,C 90.000,E1 185.106} C_DIS
LIN {X 0.040,Y -396.440,Z 989.825,A 0.000,B 0.000,C 90.000,E1 184.531} C_DIS
LIN {X 0.006,Y -396.542,Z 989.824,A 0.000,B 0.000,C 90.000,E1 184.359} C_DIS
LIN {X -0.140,Y -397.308,Z 989.822,A 0.000,B 0.000,C 90.000,E1 184.012} C_DIS
LIN {X 0.192,Y -398.382,Z 989.820,A 0.000,B 0.000,C 90.000,E1 183.612} C_DIS
LIN {X 0.020,Y -400.857,Z 989.817,A 0.000,B 0.000,C 90.000,E1 183.037} C_DIS
LIN {X -0.072,Y -405.046,Z 989.813,A 0.000,B 0.000,C 90.000,E1 182.350} C_DIS
LIN {X -0.088,Y -406.184,Z 989.812,A 0.000,B 0.000,C 90.000,E1 182.178} C_DIS
LIN {X 0.068,Y -413.290,Z 989.807,A 0.000,B 0.000,C 90.000,E1 181.318} C_DIS
LIN {X -0.038,Y -420.355,Z 989.803,A 0.000,B 0.000,C 90.000,E1 180.573} C_DIS
LIN {X 0.151,Y -432.120,Z 989.797,A 0.000,B 0.000,C 90.000,E1 179.370} C_DIS
LIN {X -0.211,Y -439.353,Z 989.793,A 0.000,B 0.000,C 90.000,E1 178.682} C_DIS
LIN {X 0.216,Y -449.393,Z 989.787,A 0.000,B 0.000,C 90.000,E1 177.593} C_DIS
LIN {X -0.170,Y -456.457,Z 989.783,A 0.000,B 0.000,C 90.000,E1 176.906} C_DIS
LIN {X 0.044,Y -461.953,Z 989.779,A 0.000,B 0.000,C 90.000,E1 176.274} C_DIS
LIN {X 0.206,Y -469.642,Z 989.774,A 0.000,B 0.000,C 90.000,E1 175.355} C_DIS
LIN {X -0.034,Y -476.168,Z 989.770,A 0.000,B 0.000,C 90.000,E1 174.609} C_DIS
LIN {X 0.050,Y -484.502,Z 989.764,A 0.000,B 0.000,C 90.000,E1 173.514} C_DIS
LIN {X -0.252,Y -491.290,Z 989.759,A 0.000,B 0.000,C 90.000,E1 172.648} C_DIS
LIN {X -0.243,Y -499.950,Z 989.752,A 0.000,B 0.000,C 90.000,E1 171.432} C_DIS
LIN {X 0.163,Y -509.148,Z 989.745,A 0.000,B 0.000,C 90.000,E1 170.038} C_DIS
LIN {X -0.264,Y -516.016,Z 989.739,A 0.000,B 0.000,C 90.000,E1 169.050} C_DIS
LIN {X 0.206,Y -523.396,Z 989.733,A 0.000,B 0.000,C 90.000,E1 167.825} C_DIS
LIN {X 0.060,Y -529.628,Z 989.727,A 0.000,B 0.000,C 90.000,E1 166.825} C_DIS
LIN {X 0.172,Y -537.479,Z 989.720,A 0.000,B 0.000,C 90.000,E1 165.519} C_DIS
LIN {X 0.205,Y -543.392,Z 989.714,A 0.000,B 0.000,C 90.000,E1 164.519} C_DIS
LIN {X 0.275,Y -552.368,Z 989.706,A 0.000,B 0.000,C 90.000,E1 162.960} C_DIS
LIN {X 0.120,Y -562.356,Z 989.695,A 0.000,B 0.000,C 90.000,E1 161.167} C_DIS
LIN {X 0.254,Y -567.469,Z 989.690,A 0.000,B 0.000,C 90.000,E1 160.188} C_DIS
LIN {X 0.283,Y -573.800,Z 989.683,A 0.000,B 0.000,C 90.000,E1 158.954} C_DIS
LIN {X -0.261,Y -579.105,Z 989.677,A 0.000,B 0.000,C 90.000,E1 157.922} C_DIS
LIN {X 0.168,Y -584.566,Z 989.671,A 0.000,B 0.000,C 90.000,E1 156.666} C_DIS
LIN {X -0.321,Y -586.957,Z 989.668,A 0.000,B 0.000,C 90.000,E1 156.177} C_DIS
LIN {X -0.251,Y -591.327,Z 989.662,A 0.000,B 0.000,C 90.000,E1 155.101} C_DIS
LIN {X -0.118,Y -595.281,Z 989.656,A 0.000,B 0.000,C 90.000,E1 154.024} C_DIS
LIN {X 0.066,Y -598.842,Z 989.650,A 0.000,B 0.000,C 90.000,E1 152.948} C_DIS
LIN {X 0.112,Y -601.337,Z 989.645,A 0.000,B 0.000,C 90.000,E1 152.153} C_DIS
LIN {X 0.069,Y -605.247,Z 989.638,A 0.000,B 0.000,C 90.000,E1 150.845} C_DIS
LIN {X 0.141,Y -608.330,Z 989.632,A 0.000,B 0.000,C 90.000,E1 149.793} C_DIS
LIN {X -0.319,Y -612.096,Z 989.625,A 0.000,B 0.000,C 90.000,E1 148.535} C_DIS
LIN {X 0.115,Y -615.838,Z 989.618,A 0.000,B 0.000,C 90.000,E1 147.199} C_DIS
LIN {X -0.342,Y -621.710,Z 989.606,A 0.000,B 0.000,C 90.000,E1 145.182} C_DIS
LIN {X -0.090,Y -626.148,Z 989.598,A 0.000,B 0.000,C 90.000,E1 143.623} C_DIS
LIN {X -0.247,Y -630.524,Z 989.589,A 0.000,B 0.000,C 90.000,E1 142.110} C_DIS
LIN {X 0.076,Y -634.841,Z 989.581,A 0.000,B 0.000,C 90.000,E1 140.561} C_DIS
LIN {X 0.100,Y -638.360,Z 989.574,A 0.000,B 0.000,C 90.000,E1 139.299} C_DIS
LIN {X 0.083,Y -642.464,Z 989.566,A 0.000,B 0.000,C 90.000,E1 137.796} C_DIS
LIN {X 0.033,Y -647.517,Z 989.556,A 0.000,B 0.000,C 90.000,E1 136.053} C_DIS
LIN {X -0.020,Y -655.240,Z 989.542,A 0.000,B 0.000,C 90.000,E1 133.581} C_DIS
LIN {X 0.241,Y -661.092,Z 989.533,A 0.000,B 0.000,C 90.000,E1 131.838} C_DIS
LIN {X 0.189,Y -666.325,Z 989.524,A 0.000,B 0.000,C 90.000,E1 130.378} C_DIS
LIN {X -0.200,Y -670.504,Z 989.518,A 0.000,B 0.000,C 90.000,E1 129.197} C_DIS
LIN {X 0.006,Y -674.361,Z 989.511,A 0.000,B 0.000,C 90.000,E1 127.971} C_DIS
LIN {X 0.142,Y -677.325,Z 989.506,A 0.000,B 0.000,C 90.000,E1 126.996} C_DIS
LIN {X 0.054,Y -680.815,Z 989.499,A 0.000,B 0.000,C 90.000,E1 125.804} C_DIS
LIN {X 0.027,Y -684.250,Z 989.492,A 0.000,B 0.000,C 90.000,E1 124.612} C_DIS
LIN {X 0.047,Y -687.462,Z 989.486,A 0.000,B 0.000,C 90.000,E1 123.420} C_DIS
LIN {X 0.179,Y -691.767,Z 989.477,A 0.000,B 0.000,C 90.000,E1 121.750} C_DIS
LIN {X 0.289,Y -694.164,Z 989.471,A 0.000,B 0.000,C 90.000,E1 120.797} C_DIS
LIN {X -0.177,Y -695.764,Z 989.467,A 0.000,B 0.000,C 90.000,E1 120.129} C_DIS
LIN {X -0.027,Y -697.163,Z 989.463,A 0.000,B 0.000,C 90.000,E1 119.411} C_DIS
LIN {X 0.140,Y -698.346,Z 989.460,A 0.000,B 0.000,C 90.000,E1 118.693} C_DIS
LIN {X 0.319,Y -699.216,Z 989.456,A 0.000,B 0.000,C 90.000,E1 117.975} C_DIS
LIN {X -0.117,Y -699.856,Z 989.452,A 0.000,B 0.000,C 90.000,E1 117.308} C_DIS
LIN {X -0.059,Y -701.106,Z 989.444,A 0.000,B 0.000,C 90.000,E1 115.899} C_DIS
LIN {X 0.186,Y -701.486,Z 989.441,A 0.000,B 0.000,C 90.000,E1 115.412} C_DIS
LIN {X -0.279,Y -701.746,Z 989.436,A 0.000,B 0.000,C 90.000,E1 114.515} C_DIS
LIN {X -0.005,Y -701.799,Z 989.435,A 0.000,B 0.000,C 90.000,E1 114.259} C_DIS
LIN {X 0.257,Y -701.429,Z 989.432,A 0.000,B 0.000,C 90.000,E1 113.770} C_DIS
LIN {X -0.112,Y -701.143,Z 989.431,A 0.000,B 0.000,C 90.000,E1 113.567} C_DIS
LIN {X 0.150,Y -699.271,Z 989.428,A 0.000,B 0.000,C 90.000,E1 113.078} C_DIS
LIN {X 0.144,Y -698.111,Z 989.427,A 0.000,B 0.000,C 90.000,E1 112.845} C_DIS
LIN {X -0.368,Y -697.143,Z 989.426,A 0.000,B 0.000,C 90.000,E1 112.770} C_DIS
LIN {X 0.035,Y -692.136,Z 989.424,A 0.000,B 0.000,C 90.000,E1 112.280} C_DIS
LIN {X 0.216,Y -690.412,Z 989.423,A 0.000,B 0.000,C 90.000,E1 112.153} C_DIS
LIN {X 0.115,Y -685.361,Z 989.422,A 0.000,B 0.000,C 90.000,E1 111.972} C_DIS
LIN {X 0.284,Y -683.033,Z 989.422,A 0.000,B 0.000,C 90.000,E1 111.897} C_DIS
LIN {X 0.196,Y -675.442,Z 989.421,A 0.000,B 0.000,C 90.000,E1 111.770} C_DIS
LIN {X 0.093,Y -671.438,Z 989.421,A 0.000,B 0.000,C 90.000,E1 111.770} C_DIS
LIN {X 0.048,Y -621.468,Z 989.421,A 0.000,B 0.000,C 90.000,E1 111.770} C_DIS
LIN {X -0.075,Y -616.073,Z 989.420,A 0.000,B 0.000,C 90.000,E1 111.663} C_DIS
LIN {X 0.137,Y -610.522,Z 989.419,A 0.000,B 0.000,C 90.000,E1 111.482} C_DIS
LIN {X 0.047,Y -602.114,Z 989.418,A 0.000,B 0.000,C 90.000,E1 111.153} C_DIS
LIN {X -0.019,Y -596.494,Z 989.416,A 0.000,B 0.000,C 90.000,E1 110.844} C_DIS
LIN {X 0.024,Y -589.395,Z 989.413,A 0.000,B 0.000,C 90.000,E1 110.355} C_DIS
LIN {X 0.190,Y -578.103,Z 989.408,A 0.000,B 0.000,C 90.000,E1 109.450} C_DIS
LIN {X -0.109,Y -573.691,Z 989.406,A 0.000,B 0.000,C 90.000,E1 109.141} C_DIS
LIN {X 0.171,Y -565.359,Z 989.403,A 0.000,B 0.000,C 90.000,E1 108.598} C_DIS
LIN {X 0.065,Y -556.650,Z 989.401,A 0.000,B 0.000,C 90.000,E1 108.181} C_DIS
LIN {X -0.126,Y -551.129,Z 989.400,A 0.000,B 0.000,C 90.000,E1 107.928} C_DIS
LIN {X 0.334,Y -549.357,Z 989.399,A 0.000,B 0.000,C 90.000,E1 107.692} C_DIS
LIN {X 0.293,Y -549.338,Z 989.398,A 0.000,B 0.000,C 90.000,E1 107.692} C_DIS
LIN {X 0.178,Y -548.818,Z 989.397,A 0.000,B 0.000,C 90.000,E1 107.402} C_DIS
LIN {X -0.137,Y -548.944,Z 989.393,A 0.000,B 0.000,C 90.000,E1 106.732} C_DIS
LIN {X -0.023,Y -549.577,Z 989.385,A 0.000,B 0.000,C 90.000,E1 105.315} C_DIS
LIN {X 0.042,Y -550.763,Z 989.373,A 0.000,B 0.000,C 90.000,E1 103.063} C_DIS
LIN {X 0.130,Y -553.180,Z 989.357,A 0.000,B 0.000,C 90.000,E1 100.254} C_DIS
LIN {X -0.277,Y -555.223,Z 989.346,A 0.000,B 0.000,C 90.000,E1 98.341} C_DIS
LIN {X 0.281,Y -556.710,Z 989.339,A 0.000,B 0.000,C 90.000,E1 96.891} C_DIS
LIN {X 0.106,Y -557.758,Z 989.332,A 0.000,B 0.000,C 90.000,E1 95.796} C_DIS
LIN {X 0.022,Y -558.742,Z 989.325,A 0.000,B 0.000,C 90.000,E1 94.416} C_DIS
LIN {X -0.252,Y -559.229,Z 989.320,A 0.000,B 0.000,C 90.000,E1 93.612} C_DIS
LIN {X -0.254,Y -560.113,Z 989.311,A 0.000,B 0.000,C 90.000,E1 91.949} C_DIS
LIN {X -0.237,Y -561.007,Z 989.302,A 0.000,B 0.000,C 90.000,E1 90.286} C_DIS
LIN {X 0.248,Y -561.588,Z 989.294,A 0.000,B 0.000,C 90.000,E1 88.854} C_DIS
LIN {X 0.192,Y -561.897,Z 989.286,A 0.000,B 0.000,C 90.000,E1 87.478} C_DIS
LIN {X -0.194,Y -562.216,Z 989.275,A 0.000,B 0.000,C 90.000,E1 85.584} C_DIS
LIN {X -0.202,Y -562.398,Z 989.268,A 0.000,B 0.000,C 90.000,E1 84.204} C_DIS
LIN {X 0.082,Y -562.730,Z 989.257,A 0.000,B 0.000,C 90.000,E1 82.243} C_DIS
LIN {X -0.108,Y -563.242,Z 989.246,A 0.000,B 0.000,C 90.000,E1 80.330} C_DIS
LIN {X -0.195,Y -564.059,Z 989.236,A 0.000,B 0.000,C 90.000,E1 78.409} C_DIS
LIN {X -0.189,Y -564.913,Z 989.226,A 0.000,B 0.000,C 90.000,E1 76.756} C_DIS
LIN {X -0.206,Y -566.542,Z 989.213,A 0.000,B 0.000,C 90.000,E1 74.283} C_DIS
LIN {X 0.167,Y -567.747,Z 989.203,A 0.000,B 0.000,C 90.000,E1 72.598} C_DIS
LIN {X 0.036,Y -568.905,Z 989.194,A 0.000,B 0.000,C 90.000,E1 70.967} C_DIS
LIN {X -0.082,Y -569.894,Z 989.185,A 0.000,B 0.000,C 90.000,E1 69.337} C_DIS
LIN {X 0.217,Y -570.717,Z 989.176,A 0.000,B 0.000,C 90.000,E1 67.667} C_DIS
LIN {X 0.180,Y -571.347,Z 989.169,A 0.000,B 0.000,C 90.000,E1 66.305} C_DIS
LIN {X 0.212,Y -571.957,Z 989.159,A 0.000,B 0.000,C 90.000,E1 64.665} C_DIS
LIN {X -0.004,Y -572.389,Z 989.150,A 0.000,B 0.000,C 90.000,E1 63.050} C_DIS
LIN {X -0.040,Y -572.725,Z 989.143,A 0.000,B 0.000,C 90.000,E1 61.691} C_DIS
LIN {X -0.078,Y -573.014,Z 989.135,A 0.000,B 0.000,C 90.000,E1 60.333} C_DIS
LIN {X 0.163,Y -573.247,Z 989.128,A 0.000,B 0.000,C 90.000,E1 58.948} C_DIS
LIN {X 0.041,Y -573.438,Z 989.119,A 0.000,B 0.000,C 90.000,E1 57.327} C_DIS
LIN {X 0.276,Y -573.548,Z 989.112,A 0.000,B 0.000,C 90.000,E1 56.215} C_DIS
LIN {X -0.137,Y -573.595,Z 989.105,A 0.000,B 0.000,C 90.000,E1 54.895} C_DIS
LIN {X 0.242,Y -573.339,Z 989.097,A 0.000,B 0.000,C 90.000,E1 53.497} C_DIS
LIN {X 0.006,Y -572.928,Z 989.091,A 0.000,B 0.000,C 90.000,E1 52.431} C_DIS
LIN {X -0.026,Y -572.539,Z 989.087,A 0.000,B 0.000,C 90.000,E1 51.618} C_DIS
LIN {X 0.078,Y -571.807,Z 989.081,A 0.000,B 0.000,C 90.000,E1 50.517} C_DIS
LIN {X 0.036,Y -571.168,Z 989.076,A 0.000,B 0.000,C 90.000,E1 49.703} C_DIS
LIN {X 0.054,Y -570.072,Z 989.070,A 0.000,B 0.000,C 90.000,E1 48.609} C_DIS
LIN {X -0.316,Y -568.737,Z 989.064,A 0.000,B 0.000,C 90.000,E1 47.553} C_DIS
LIN {X -0.018,Y -567.523,Z 989.060,A 0.000,B 0.000,C 90.000,E1 46.701} C_DIS
LIN {X -0.050,Y -565.641,Z 989.053,A 0.000,B 0.000,C 90.000,E1 45.607} C_DIS
LIN {X 0.203,Y -563.999,Z 989.049,A 0.000,B 0.000,C 90.000,E1 44.757} C_DIS
LIN {X 0.042,Y -562.134,Z 989.044,A 0.000,B 0.000,C 90.000,E1 43.947} C_DIS
LIN {X -0.141,Y -559.989,Z 989.040,A 0.000,B 0.000,C 90.000,E1 43.137} C_DIS
LIN {X 0.060,Y -557.571,Z 989.035,A 0.000,B 0.000,C 90.000,E1 42.285} C_DIS
